gfCNCPoint5[14448] = {X 306.6871, Y 54.0357, Z -7.1667, A 0.000, B 0.000, C 0.000 }
gfCNCPoint5[14449] = {X 307.6171, Y 53.7103, Z -7.1667, A 0.000, B 0.000, C 0.000 }
gfCNCPoint5[14450] = {X 308.5962, Y 53.6000, Z -7.1667, A 0.000, B 0.000, C 0.000 }
gfCNCPoint5[14451] = {X 324.3107, Y 53.6000, Z -7.1667, A 0.000, B 0.000, C 0.000 }
gfCNCPoint5[14452] = {X 325.2898, Y 53.7103, Z -7.1667, A 0.000, B 0.000, C 0.000 }
gfCNCPoint5[14453] = {X 326.2198, Y 54.0357, Z -7.1667, A 0.000, B 0.000, C 0.000 }
gfCNCPoint5[14454] = {X 327.0540, Y 54.5599, Z -7.1667, A 0.000, B 0.000, C 0.000 }
gfCNCPoint5[14455] = {X 327.7507, Y 55.2566, Z -7.1667, A 0.000, B 0.000, C 0.000 }
gfCNCPoint5[14456] = {X 328.2750, Y 56.0909, Z -7.1667, A 0.000, B 0.000, C 0.000 }
gfCNCPoint5[14457] = {X 328.6004, Y 57.0209, Z -7.1667, A 0.000, B 0.000, C 0.000 }
gfCNCPoint5[14458] = {X 328.7107, Y 58.0000, Z -7.1667, A 0.000, B 0.000, C 0.000 }
gfCNCPoint5[14459] = {X 328.7107, Y 58.9362, Z -7.1667, A 0.000, B 0.000, C 0.000 }
gfCNCPoint5[14460] = {X 328.6172, Y 59.8190, Z -7.1667, A 0.000, B 0.000, C 0.000 }
gfCNCPoint5[14461] = {X 328.3499, Y 60.6656, Z -7.1667, A 0.000, B 0.000, C 0.000 }
gfCNCPoint5[14462] = {X 327.9194, Y 61.4419, Z -7.1667, A 0.000, B 0.000, C 0.000 }
gfCNCPoint5[14463] = {X 327.3430, Y 62.1171, Z -7.1667, A 0.000, B 0.000, C 0.000 }
gfCNCPoint5[14464] = {X 326.6437, Y 62.6640, Z -7.1667, A 0.000, B 0.000, C 0.000 }
gfCNCPoint5[14465] = {X 325.8496, Y 63.0607, Z -7.1667, A 0.000, B 0.000, C 0.000 }
gfCNCPoint5[14466] = {X 324.9923, Y 63.2915, Z -7.1667, A 0.000, B 0.000, C 0.000 }
gfCNCPoint5[14467] = {X 324.9942, Y 83.2293, Z -7.1667, A 0.000, B 0.000, C 0.000 }
gfCNCPoint5[14468] = {X 325.0078, Y 84.6142, Z -7.1667, A 0.000, B 0.000, C 0.000 }
gfCNCPoint5[14469] = {X 325.0827, Y 85.8241, Z -7.1667, A 0.000, B 0.000, C 0.000 }
gfCNCPoint5[14470] = {X 325.2965, Y 87.0173, Z -7.1667, A 0.000, B 0.000, C 0.000 }
gfCNCPoint5[14471] = {X 325.7310, Y 87.4224, Z -7.1667, A 0.000, B 0.000, C 0.000 }
gfCNCPoint5[14472] = {X 326.2477, Y 87.7156, Z -7.1667, A 0.000, B 0.000, C 0.000 }
gfCNCPoint5[14473] = {X 328.0176, Y 88.4226, Z -7.1667, A 0.000, B 0.000, C 0.000 }
gfCNCPoint5[14474] = {X 329.8594, Y 88.9123, Z -7.1667, A 0.000, B 0.000, C 0.000 }
gfCNCPoint5[14475] = {X 332.9373, Y 89.4644, Z -7.1667, A 0.000, B 0.000, C 0.000 }
gfCNCPoint5[14476] = {X 336.0431, Y 89.8280, Z -7.1667, A 0.000, B 0.000, C 0.000 }
gfCNCPoint5[14477] = {X 340.4120, Y 90.1221, Z -7.1667, A 0.000, B 0.000, C 0.000 }
gfCNCPoint5[14478] = {X 344.7882, Y 90.2759, Z -7.1667, A 0.000, B 0.000, C 0.000 }
gfCNCPoint5[14479] = {X 349.1670, Y 90.2890, Z -7.1667, A 0.000, B 0.000, C 0.000 }
gfCNCPoint5[14480] = {X 353.3143, Y 90.2206, Z -7.1667, A 0.000, B 0.000, C 0.000 }
gfCNCPoint5[14481] = {X 357.4564, Y 90.0018, Z -7.1667, A 0.000, B 0.000, C 0.000 }
gfCNCPoint5[14482] = {X 361.5878, Y 89.6328, Z -7.1667, A 0.000, B 0.000, C 0.000 }
gfCNCPoint5[14483] = {X 363.6656, Y 89.3462, Z -7.1667, A 0.000, B 0.000, C 0.000 }
gfCNCPoint5[14484] = {X 365.7243, Y 88.9447, Z -7.1667, A 0.000, B 0.000, C 0.000 }
gfCNCPoint5[14485] = {X 367.7576, Y 88.4298, Z -7.1667, A 0.000, B 0.000, C 0.000 }
gfCNCPoint5[14486] = {X 368.6806, Y 88.1197, Z -7.1667, A 0.000, B 0.000, C 0.000 }
gfCNCPoint5[14487] = {X 369.5629, Y 87.7078, Z -7.1667, A 0.000, B 0.000, C 0.000 }
gfCNCPoint5[14488] = {X 370.3933, Y 87.1992, Z -7.1667, A 0.000, B 0.000, C 0.000 }
gfCNCPoint5[14489] = {X 370.5198, Y 87.0673, Z -7.1667, A 0.000, B 0.000, C 0.000 }
gfCNCPoint5[14490] = {X 370.5851, Y 86.8966, Z -7.1667, A 0.000, B 0.000, C 0.000 }
gfCNCPoint5[14491] = {X 370.7755, Y 85.3680, Z -7.1667, A 0.000, B 0.000, C 0.000 }
gfCNCPoint5[14492] = {X 370.8391, Y 83.8288, Z -7.1667, A 0.000, B 0.000, C 0.000 }
gfCNCPoint5[14493] = {X 370.8379, Y 63.2810, Z -7.1667, A 0.000, B 0.000, C 0.000 }
gfCNCPoint5[14494] = {X 369.9788, Y 63.0556, Z -7.1667, A 0.000, B 0.000, C 0.000 }
gfCNCPoint5[14495] = {X 369.1826, Y 62.6623, Z -7.1667, A 0.000, B 0.000, C 0.000 }
gfCNCPoint5[14496] = {X 368.4815, Y 62.1171, Z -7.1667, A 0.000, B 0.000, C 0.000 }
gfCNCPoint5[14497] = {X 367.9042, Y 61.4423, Z -7.1667, A 0.000, B 0.000, C 0.000 }
gfCNCPoint5[14498] = {X 367.4741, Y 60.6652, Z -7.1667, A 0.000, B 0.000, C 0.000 }
gfCNCPoint5[14499] = {X 367.2089, Y 59.8176, Z -7.1667, A 0.000, B 0.000, C 0.000 }
gfCNCPoint5[14500] = {X 367.1193, Y 58.9341, Z -7.1667, A 0.000, B 0.000, C 0.000 }
gfCNCPoint5[14501] = {X 367.1193, Y 58.0000, Z -7.1667, A 0.000, B 0.000, C 0.000 }
gfCNCPoint5[14502] = {X 367.2296, Y 57.0209, Z -7.1667, A 0.000, B 0.000, C 0.000 }
gfCNCPoint5[14503] = {X 367.5550, Y 56.0909, Z -7.1667, A 0.000, B 0.000, C 0.000 }
gfCNCPoint5[14504] = {X 368.0792, Y 55.2566, Z -7.1667, A 0.000, B 0.000, C 0.000 }
gfCNCPoint5[14505] = {X 368.7759, Y 54.5599, Z -7.1667, A 0.000, B 0.000, C 0.000 }
gfCNCPoint5[14506] = {X 369.6102, Y 54.0357, Z -7.1667, A 0.000, B 0.000, C 0.000 }
gfCNCPoint5[14507] = {X 370.5402, Y 53.7103, Z -7.1667, A 0.000, B 0.000, C 0.000 }
gfCNCPoint5[14508] = {X 371.5193, Y 53.6000, Z -7.1667, A 0.000, B 0.000, C 0.000 }
gfCNCPoint5[14509] = {X 388.0597, Y 53.6000, Z -7.1667, A 0.000, B 0.000, C 0.000 }
gfCNCPoint5[14510] = {X 389.0388, Y 53.7103, Z -7.1667, A 0.000, B 0.000, C 0.000 }
gfCNCPoint5[14511] = {X 389.9688, Y 54.0357, Z -7.1667, A 0.000, B 0.000, C 0.000 }
gfCNCPoint5[14512] = {X 390.8030, Y 54.5599, Z -7.1667, A 0.000, B 0.000, C 0.000 }
gfCNCPoint5[14513] = {X 391.4997, Y 55.2566, Z -7.1667, A 0.000, B 0.000, C 0.000 }
gfCNCPoint5[14514] = {X 392.0239, Y 56.0909, Z -7.1667, A 0.000, B 0.000, C 0.000 }
gfCNCPoint5[14515] = {X 392.3494, Y 57.0209, Z -7.1667, A 0.000, B 0.000, C 0.000 }
gfCNCPoint5[14516] = {X 392.4597, Y 58.0000, Z -7.1667, A 0.000, B 0.000, C 0.000 }
gfCNCPoint5[14517] = {X 392.4595, Y 58.9704, Z -7.1667, A 0.000, B 0.000, C 0.000 }
gfCNCPoint5[14518] = {X 392.3419, Y 59.9454, Z -7.1667, A 0.000, B 0.000, C 0.000 }
gfCNCPoint5[14519] = {X 392.0109, Y 60.8701, Z -7.1667, A 0.000, B 0.000, C 0.000 }
gfCNCPoint5[14520] = {X 391.5686, Y 61.5895, Z -7.1667, A 0.000, B 0.000, C 0.000 }
gfCNCPoint5[14521] = {X 390.9977, Y 62.2117, Z -7.1667, A 0.000, B 0.000, C 0.000 }
gfCNCPoint5[14522] = {X 390.3190, Y 62.7141, Z -7.1667, A 0.000, B 0.000, C 0.000 }
gfCNCPoint5[14523] = {X 389.5572, Y 63.0784, Z -7.1667, A 0.000, B 0.000, C 0.000 }
gfCNCPoint5[14524] = {X 388.7400, Y 63.2913, Z -7.1667, A 0.000, B 0.000, C 0.000 }
gfCNCPoint5[14525] = {X 388.7400, Y 83.9247, Z -7.1667, A 0.000, B 0.000, C 0.000 }
gfCNCPoint5[14526] = {X 388.7379, Y 84.6149, Z -7.1667, A 0.000, B 0.000, C 0.000 }
gfCNCPoint5[14527] = {X 388.6777, Y 86.2800, Z -7.1667, A 0.000, B 0.000, C 0.000 }
gfCNCPoint5[14528] = {X 388.4725, Y 87.9334, Z -7.1667, A 0.000, B 0.000, C 0.000 }
gfCNCPoint5[14529] = {X 388.1239, Y 89.5626, Z -7.1667, A 0.000, B 0.000, C 0.000 }
gfCNCPoint5[14530] = {X 387.5878, Y 91.1605, Z -7.1667, A 0.000, B 0.000, C 0.000 }
gfCNCPoint5[14531] = {X 386.8330, Y 92.6676, Z -7.1667, A 0.000, B 0.000, C 0.000 }
gfCNCPoint5[14532] = {X 385.8745, Y 94.0540, Z -7.1667, A 0.000, B 0.000, C 0.000 }
gfCNCPoint5[14533] = {X 384.7313, Y 95.2924, Z -7.1667, A 0.000, B 0.000, C 0.000 }
gfCNCPoint5[14534] = {X 383.5035, Y 96.3481, Z -7.1667, A 0.000, B 0.000, C 0.000 }
gfCNCPoint5[14535] = {X 382.1889, Y 97.2937, Z -7.1667, A 0.000, B 0.000, C 0.000 }
gfCNCPoint5[14536] = {X 382.4521, Y 97.6951, Z -7.1667, A 0.000, B 0.000, C 0.000 }
gfCNCPoint5[14537] = {X 391.5259, Y 97.6951, Z -7.1667, A 0.000, B 0.000, C 0.000 }
gfCNCPoint5[14538] = {X 391.5259, Y 97.0659, Z -7.1667, A 0.000, B 0.000, C 0.000 }
gfCNCPoint5[14539] = {X 391.6193, Y 96.1159, Z -7.1667, A 0.000, B 0.000, C 0.000 }
gfCNCPoint5[14540] = {X 391.8959, Y 95.2021, Z -7.1667, A 0.000, B 0.000, C 0.000 }
gfCNCPoint5[14541] = {X 392.3450, Y 94.3598, Z -7.1667, A 0.000, B 0.000, C 0.000 }
gfCNCPoint5[14542] = {X 392.9496, Y 93.6209, Z -7.1667, A 0.000, B 0.000, C 0.000 }
gfCNCPoint5[14543] = {X 393.6864, Y 93.0139, Z -7.1667, A 0.000, B 0.000, C 0.000 }
gfCNCPoint5[14544] = {X 394.5273, Y 92.5620, Z -7.1667, A 0.000, B 0.000, C 0.000 }
gfCNCPoint5[14545] = {X 395.4401, Y 92.2825, Z -7.1667, A 0.000, B 0.000, C 0.000 }
gfCNCPoint5[14546] = {X 396.3899, Y 92.1860, Z -7.1667, A 0.000, B 0.000, C 0.000 }
gfCNCPoint5[14547] = {X 397.3090, Y 92.1443, Z -7.1667, A 0.000, B 0.000, C 0.000 }
gfCNCPoint5[14548] = {X 398.2250, Y 92.0575, Z -7.1667, A 0.000, B 0.000, C 0.000 }
gfCNCPoint5[14549] = {X 398.7531, Y 91.9291, Z -7.1667, A 0.000, B 0.000, C 0.000 }
gfCNCPoint5[14550] = {X 399.2394, Y 91.6865, Z -7.1667, A 0.000, B 0.000, C 0.000 }
gfCNCPoint5[14551] = {X 426.8261, Y 74.0196, Z -7.1667, A 0.000, B 0.000, C 0.000 }
gfCNCPoint5[14552] = {X 403.5510, Y 64.8882, Z -7.1667, A 0.000, B 0.000, C 0.000 }
gfCNCPoint5[14553] = {X 402.0098, Y 64.3725, Z -7.1667, A 0.000, B 0.000, C 0.000 }
gfCNCPoint5[14554] = {X 400.4236, Y 64.0186, Z -7.1667, A 0.000, B 0.000, C 0.000 }
gfCNCPoint5[14555] = {X 398.8190, Y 73.4835, Z -7.1667, A 0.000, B 0.000, C 0.000 }
gfCNCPoint5[14556] = {X 398.8183, Y 80.5563, Z -7.1667, A 0.000, B 0.000, C 0.000 }
gfCNCPoint5[14557] = {X 405.8022, Y 76.0837, Z -7.1667, A 0.000, B 0.000, C 0.000 }
gfCNCPoint5[14558] = {X 400.0393, Y 73.8228, Z -7.1667, A 0.000, B 0.000, C 0.000 }
gfCNCPoint5[14559] = {X 399.4379, Y 73.6216, Z -7.1667, A 0.000, B 0.000, C 0.000 }
gfCNCPoint5[14560] = {X 398.8190, Y 73.4835, Z -7.1667, A 0.000, B 0.000, C 0.000 }
gfCNCPoint5[14561] = {X 399.2202, Y 71.1173, Z -7.1667, A 0.000, B 0.000, C 0.000 }
gfCNCPoint5[14562] = {X 398.7493, Y 71.0509, Z -7.1667, A 0.000, B 0.000, C 0.000 }
gfCNCPoint5[14563] = {X 398.2755, Y 71.0108, Z -7.1667, A 0.000, B 0.000, C 0.000 }
gfCNCPoint5[14564] = {X 397.3438, Y 70.9529, Z -7.1667, A 0.000, B 0.000, C 0.000 }
gfCNCPoint5[14565] = {X 396.4193, Y 70.8233, Z -7.1667, A 0.000, B 0.000, C 0.000 }
gfCNCPoint5[14566] = {X 396.4180, Y 84.5897, Z -7.1667, A 0.000, B 0.000, C 0.000 }
gfCNCPoint5[14567] = {X 396.4178, Y 84.9436, Z -7.1667, A 0.000, B 0.000, C 0.000 }
gfCNCPoint5[14568] = {X 411.0581, Y 75.5677, Z -7.1667, A 0.000, B 0.000, C 0.000 }
gfCNCPoint5[14569] = {X 400.9172, Y 71.5892, Z -7.1667, A 0.000, B 0.000, C 0.000 }
gfCNCPoint5[14570] = {X 400.0809, Y 71.3094, Z -7.1667, A 0.000, B 0.000, C 0.000 }
gfCNCPoint5[14571] = {X 399.2202, Y 71.1173, Z -7.1667, A 0.000, B 0.000, C 0.000 }
gfCNCPoint5[14572] = {X 399.6213, Y 68.7510, Z -7.1667, A 0.000, B 0.000, C 0.000 }
gfCNCPoint5[14573] = {X 398.9961, Y 68.6635, Z -7.1667, A 0.000, B 0.000, C 0.000 }
gfCNCPoint5[14574] = {X 398.3668, Y 68.6122, Z -7.1667, A 0.000, B 0.000, C 0.000 }
gfCNCPoint5[14575] = {X 397.6025, Y 68.5668, Z -7.1667, A 0.000, B 0.000, C 0.000 }
gfCNCPoint5[14576] = {X 396.8441, Y 68.4612, Z -7.1667, A 0.000, B 0.000, C 0.000 }
gfCNCPoint5[14577] = {X 395.3939, Y 68.0824, Z -7.1667, A 0.000, B 0.000, C 0.000 }
gfCNCPoint5[14578] = {X 394.0196, Y 67.4844, Z -7.1667, A 0.000, B 0.000, C 0.000 }
gfCNCPoint5[14579] = {X 394.0180, Y 84.5973, Z -7.1667, A 0.000, B 0.000, C 0.000 }
gfCNCPoint5[14580] = {X 394.0185, Y 84.7621, Z -7.1667, A 0.000, B 0.000, C 0.000 }
gfCNCPoint5[14581] = {X 394.0179, Y 84.9270, Z -7.1667, A 0.000, B 0.000, C 0.000 }
gfCNCPoint5[14582] = {X 393.9676, Y 86.3327, Z -7.1667, A 0.000, B 0.000, C 0.000 }
gfCNCPoint5[14583] = {X 393.8362, Y 87.7333, Z -7.1667, A 0.000, B 0.000, C 0.000 }
gfCNCPoint5[14584] = {X 395.0679, Y 87.4789, Z -7.1667, A 0.000, B 0.000, C 0.000 }
gfCNCPoint5[14585] = {X 396.3222, Y 87.3863, Z -7.1667, A 0.000, B 0.000, C 0.000 }
gfCNCPoint5[14586] = {X 396.7204, Y 87.3714, Z -7.1667, A 0.000, B 0.000, C 0.000 }
gfCNCPoint5[14587] = {X 397.1179, Y 87.3452, Z -7.1667, A 0.000, B 0.000, C 0.000 }
gfCNCPoint5[14588] = {X 416.3141, Y 75.0517, Z -7.1667, A 0.000, B 0.000, C 0.000 }
gfCNCPoint5[14589] = {X 401.7952, Y 69.3555, Z -7.1667, A 0.000, B 0.000, C 0.000 }
gfCNCPoint5[14590] = {X 400.7239, Y 68.9971, Z -7.1667, A 0.000, B 0.000, C 0.000 }
gfCNCPoint5[14591] = {X 399.6213, Y 68.7510, Z -7.1667, A 0.000, B 0.000, C 0.000 }
gfCNCPoint5[14592] = {X 400.0225, Y 66.3848, Z -7.1667, A 0.000, B 0.000, C 0.000 }
gfCNCPoint5[14593] = {X 399.2382, Y 66.2757, Z -7.1667, A 0.000, B 0.000, C 0.000 }
gfCNCPoint5[14594] = {X 398.4488, Y 66.2132, Z -7.1667, A 0.000, B 0.000, C 0.000 }
gfCNCPoint5[14595] = {X 397.3046, Y 66.1054, Z -7.1667, A 0.000, B 0.000, C 0.000 }
gfCNCPoint5[14596] = {X 396.1916, Y 65.8188, Z -7.1667, A 0.000, B 0.000, C 0.000 }
gfCNCPoint5[14597] = {X 395.1376, Y 65.3607, Z -7.1667, A 0.000, B 0.000, C 0.000 }
gfCNCPoint5[14598] = {X 394.1689, Y 64.7424, Z -7.1667, A 0.000, B 0.000, C 0.000 }
gfCNCPoint5[14599] = {X 393.3095, Y 63.9793, Z -7.1667, A 0.000, B 0.000, C 0.000 }
gfCNCPoint5[14600] = {X 392.5128, Y 64.6963, Z -7.1667, A 0.000, B 0.000, C 0.000 }
gfCNCPoint5[14601] = {X 391.6198, Y 65.2889, Z -7.1667, A 0.000, B 0.000, C 0.000 }
gfCNCPoint5[14602] = {X 391.6180, Y 84.6054, Z -7.1667, A 0.000, B 0.000, C 0.000 }
gfCNCPoint5[14603] = {X 391.5819, Y 86.0254, Z -7.1667, A 0.000, B 0.000, C 0.000 }
gfCNCPoint5[14604] = {X 391.4541, Y 87.4402, Z -7.1667, A 0.000, B 0.000, C 0.000 }
gfCNCPoint5[14605] = {X 391.2298, Y 88.8724, Z -7.1667, A 0.000, B 0.000, C 0.000 }
gfCNCPoint5[14606] = {X 390.9114, Y 90.2866, Z -7.1667, A 0.000, B 0.000, C 0.000 }
gfCNCPoint5[14607] = {X 390.3349, Y 92.0503, Z -7.1667, A 0.000, B 0.000, C 0.000 }
gfCNCPoint5[14608] = {X 389.5433, Y 93.7285, Z -7.1667, A 0.000, B 0.000, C 0.000 }
gfCNCPoint5[14609] = {X 388.5489, Y 95.2951, Z -7.1667, A 0.000, B 0.000, C 0.000 }
gfCNCPoint5[14610] = {X 389.3446, Y 95.2951, Z -7.1667, A 0.000, B 0.000, C 0.000 }
gfCNCPoint5[14611] = {X 389.7639, Y 94.0857, Z -7.1667, A 0.000, B 0.000, C 0.000 }
gfCNCPoint5[14612] = {X 390.3886, Y 92.9683, Z -7.1667, A 0.000, B 0.000, C 0.000 }
gfCNCPoint5[14613] = {X 391.1994, Y 91.9777, Z -7.1667, A 0.000, B 0.000, C 0.000 }
gfCNCPoint5[14614] = {X 392.1711, Y 91.1444, Z -7.1667, A 0.000, B 0.000, C 0.000 }
gfCNCPoint5[14615] = {X 393.2738, Y 90.4942, Z -7.1667, A 0.000, B 0.000, C 0.000 }
gfCNCPoint5[14616] = {X 394.4733, Y 90.0472, Z -7.1667, A 0.000, B 0.000, C 0.000 }
gfCNCPoint5[14617] = {X 395.4072, Y 89.8548, Z -7.1667, A 0.000, B 0.000, C 0.000 }
gfCNCPoint5[14618] = {X 396.3583, Y 89.7861, Z -7.1667, A 0.000, B 0.000, C 0.000 }
gfCNCPoint5[14619] = {X 397.1424, Y 89.7501, Z -7.1667, A 0.000, B 0.000, C 0.000 }
gfCNCPoint5[14620] = {X 397.9239, Y 89.6764, Z -7.1667, A 0.000, B 0.000, C 0.000 }
gfCNCPoint5[14621] = {X 417.6084, Y 77.0728, Z -7.1667, A 0.000, B 0.000, C 0.000 }
gfCNCPoint5[14622] = {X 421.5701, Y 74.5357, Z -7.1667, A 0.000, B 0.000, C 0.000 }
gfCNCPoint5[14623] = {X 402.6731, Y 67.1218, Z -7.1667, A 0.000, B 0.000, C 0.000 }
gfCNCPoint5[14624] = {X 401.3668, Y 66.6848, Z -7.1667, A 0.000, B 0.000, C 0.000 }
gfCNCPoint5[14625] = {X 400.0225, Y 66.3848, Z -7.1667, A 0.000, B 0.000, C 0.000 }
gfCNCPoint5[14626] = {X 400.4236, Y 64.0186, Z -7.1667, A 0.000, B 0.000, C 0.000 }
gfCNCPoint5[14627] = {X 399.4750, Y 63.8873, Z -7.1667, A 0.000, B 0.000, C 0.000 }
gfCNCPoint5[14628] = {X 398.5200, Y 63.8139, Z -7.1667, A 0.000, B 0.000, C 0.000 }
gfCNCPoint5[14629] = {X 397.5544, Y 63.7098, Z -7.1667, A 0.000, B 0.000, C 0.000 }
gfCNCPoint5[14630] = {X 396.6285, Y 63.4165, Z -7.1667, A 0.000, B 0.000, C 0.000 }
gfCNCPoint5[14631] = {X 395.7791, Y 62.9457, Z -7.1667, A 0.000, B 0.000, C 0.000 }
gfCNCPoint5[14632] = {X 395.0397, Y 62.3160, Z -7.1667, A 0.000, B 0.000, C 0.000 }
gfCNCPoint5[14633] = {X 394.4660, Y 61.5934, Z -7.1667, A 0.000, B 0.000, C 0.000 }
gfCNCPoint5[14634] = {X 394.0386, Y 60.7757, Z -7.1667, A 0.000, B 0.000, C 0.000 }
gfCNCPoint5[14635] = {X 393.7727, Y 59.8922, Z -7.1667, A 0.000, B 0.000, C 0.000 }
gfCNCPoint5[14636] = {X 393.6779, Y 58.9744, Z -7.1667, A 0.000, B 0.000, C 0.000 }
gfCNCPoint5[14637] = {X 393.6777, Y 58.0000, Z -7.1667, A 0.000, B 0.000, C 0.000 }
gfCNCPoint5[14638] = {X 393.7668, Y 57.0718, Z -7.1667, A 0.000, B 0.000, C 0.000 }
gfCNCPoint5[14639] = {X 394.0309, Y 56.1774, Z -7.1667, A 0.000, B 0.000, C 0.000 }
gfCNCPoint5[14640] = {X 394.4602, Y 55.3496, Z -7.1667, A 0.000, B 0.000, C 0.000 }
gfCNCPoint5[14641] = {X 395.0391, Y 54.6186, Z -7.1667, A 0.000, B 0.000, C 0.000 }
gfCNCPoint5[14642] = {X 395.7864, Y 53.9833, Z -7.1667, A 0.000, B 0.000, C 0.000 }
gfCNCPoint5[14643] = {X 396.6455, Y 53.5102, Z -7.1667, A 0.000, B 0.000, C 0.000 }
gfCNCPoint5[14644] = {X 397.5819, Y 53.2186, Z -7.1667, A 0.000, B 0.000, C 0.000 }
gfCNCPoint5[14645] = {X 398.5577, Y 53.1200, Z -7.1667, A 0.000, B 0.000, C 0.000 }
gfCNCPoint5[14646] = {X 419.4886, Y 53.1200, Z -7.1667, A 0.000, B 0.000, C 0.000 }
gfCNCPoint5[14647] = {X 420.5533, Y 53.2376, Z -7.1667, A 0.000, B 0.000, C 0.000 }
gfCNCPoint5[14648] = {X 421.5667, Y 53.5846, Z -7.1667, A 0.000, B 0.000, C 0.000 }
gfCNCPoint5[14649] = {X 422.4800, Y 54.1443, Z -7.1667, A 0.000, B 0.000, C 0.000 }
gfCNCPoint5[14650] = {X 423.2491, Y 54.8899, Z -7.1667, A 0.000, B 0.000, C 0.000 }
gfCNCPoint5[14651] = {X 423.8371, Y 55.7852, Z -7.1667, A 0.000, B 0.000, C 0.000 }
gfCNCPoint5[14652] = {X 424.2155, Y 56.7873, Z -7.1667, A 0.000, B 0.000, C 0.000 }
gfCNCPoint5[14653] = {X 424.3662, Y 57.8478, Z -7.1667, A 0.000, B 0.000, C 0.000 }
gfCNCPoint5[14654] = {X 429.8191, Y 59.9722, Z -7.1667, A 0.000, B 0.000, C 0.000 }
gfCNCPoint5[14655] = {X 457.2980, Y 70.8751, Z -7.1667, A 0.000, B 0.000, C 0.000 }
gfCNCPoint5[14656] = {X 457.2983, Y 63.6739, Z -7.1667, A 0.000, B 0.000, C 0.000 }
gfCNCPoint5[14657] = {X 456.2903, Y 63.3054, Z -7.1667, A 0.000, B 0.000, C 0.000 }
gfCNCPoint5[14658] = {X 455.3872, Y 62.7254, Z -7.1667, A 0.000, B 0.000, C 0.000 }
gfCNCPoint5[14659] = {X 454.6327, Y 61.9621, Z -7.1667, A 0.000, B 0.000, C 0.000 }
gfCNCPoint5[14660] = {X 454.0633, Y 61.0524, Z -7.1667, A 0.000, B 0.000, C 0.000 }
gfCNCPoint5[14661] = {X 453.7066, Y 60.0401, Z -7.1667, A 0.000, B 0.000, C 0.000 }
gfCNCPoint5[14662] = {X 453.5798, Y 58.9744, Z -7.1667, A 0.000, B 0.000, C 0.000 }
gfCNCPoint5[14663] = {X 453.5796, Y 58.0000, Z -7.1667, A 0.000, B 0.000, C 0.000 }
gfCNCPoint5[14664] = {X 453.6734, Y 57.0480, Z -7.1667, A 0.000, B 0.000, C 0.000 }
gfCNCPoint5[14665] = {X 453.9511, Y 56.1325, Z -7.1667, A 0.000, B 0.000, C 0.000 }
gfCNCPoint5[14666] = {X 454.4020, Y 55.2888, Z -7.1667, A 0.000, B 0.000, C 0.000 }
gfCNCPoint5[14667] = {X 455.0089, Y 54.5493, Z -7.1667, A 0.000, B 0.000, C 0.000 }
gfCNCPoint5[14668] = {X 455.7484, Y 53.9424, Z -7.1667, A 0.000, B 0.000, C 0.000 }
gfCNCPoint5[14669] = {X 456.5921, Y 53.4915, Z -7.1667, A 0.000, B 0.000, C 0.000 }
gfCNCPoint5[14670] = {X 457.5076, Y 53.2138, Z -7.1667, A 0.000, B 0.000, C 0.000 }
gfCNCPoint5[14671] = {X 458.4596, Y 53.1200, Z -7.1667, A 0.000, B 0.000, C 0.000 }
gfCNCPoint5[14672] = {X 475.0000, Y 53.1200, Z -7.1667, A 0.000, B 0.000, C 0.000 }
gfCNCPoint5[14673] = {X 475.9520, Y 53.2138, Z -7.1667, A 0.000, B 0.000, C 0.000 }
gfCNCPoint5[14674] = {X 476.8675, Y 53.4915, Z -7.1667, A 0.000, B 0.000, C 0.000 }
gfCNCPoint5[14675] = {X 477.7112, Y 53.9424, Z -7.1667, A 0.000, B 0.000, C 0.000 }
gfCNCPoint5[14676] = {X 478.4507, Y 54.5493, Z -7.1667, A 0.000, B 0.000, C 0.000 }
gfCNCPoint5[14677] = {X 479.0576, Y 55.2888, Z -7.1667, A 0.000, B 0.000, C 0.000 }
gfCNCPoint5[14678] = {X 479.5085, Y 56.1325, Z -7.1667, A 0.000, B 0.000, C 0.000 }
gfCNCPoint5[14679] = {X 479.7862, Y 57.0480, Z -7.1667, A 0.000, B 0.000, C 0.000 }
gfCNCPoint5[14680] = {X 479.8800, Y 58.0000, Z -7.1667, A 0.000, B 0.000, C 0.000 }
gfCNCPoint5[14681] = {X 479.8798, Y 58.9744, Z -7.1667, A 0.000, B 0.000, C 0.000 }
gfCNCPoint5[14682] = {X 479.7530, Y 60.0402, Z -7.1667, A 0.000, B 0.000, C 0.000 }
gfCNCPoint5[14683] = {X 479.3962, Y 61.0525, Z -7.1667, A 0.000, B 0.000, C 0.000 }
gfCNCPoint5[14684] = {X 478.8268, Y 61.9623, Z -7.1667, A 0.000, B 0.000, C 0.000 }
gfCNCPoint5[14685] = {X 478.0722, Y 62.7256, Z -7.1667, A 0.000, B 0.000, C 0.000 }
gfCNCPoint5[14686] = {X 477.1691, Y 63.3055, Z -7.1667, A 0.000, B 0.000, C 0.000 }
gfCNCPoint5[14687] = {X 476.1610, Y 63.6739, Z -7.1667, A 0.000, B 0.000, C 0.000 }
gfCNCPoint5[14688] = {X 476.1614, Y 92.3307, Z -7.1667, A 0.000, B 0.000, C 0.000 }
gfCNCPoint5[14689] = {X 476.3600, Y 92.3888, Z -7.1667, A 0.000, B 0.000, C 0.000 }
gfCNCPoint5[14690] = {X 476.5570, Y 92.4517, Z -7.1667, A 0.000, B 0.000, C 0.000 }
gfCNCPoint5[14691] = {X 477.4766, Y 92.8687, Z -7.1667, A 0.000, B 0.000, C 0.000 }
gfCNCPoint5[14692] = {X 478.2902, Y 93.4667, Z -7.1667, A 0.000, B 0.000, C 0.000 }
gfCNCPoint5[14693] = {X 478.9626, Y 94.2200, Z -7.1667, A 0.000, B 0.000, C 0.000 }
gfCNCPoint5[14694] = {X 479.4648, Y 95.0960, Z -7.1667, A 0.000, B 0.000, C 0.000 }
gfCNCPoint5[14695] = {X 479.7751, Y 96.0569, Z -7.1667, A 0.000, B 0.000, C 0.000 }
gfCNCPoint5[14696] = {X 479.8800, Y 97.0611, Z -7.1667, A 0.000, B 0.000, C 0.000 }
gfCNCPoint5[14697] = {X 479.8800, Y 97.6951, Z -7.1667, A 0.000, B 0.000, C 0.000 }
gfCNCPoint5[14698] = {X 479.4000, Y 97.6951, Z -7.1667, A 0.000, B 0.000, C 0.000 }
gfCNCPoint5[14699] = {X 479.4000, Y 98.0000, Z -7.1667, A 0.000, B 0.000, C 0.000 }
gfCNCPoint5[14700] = {X 479.2897, Y 98.9791, Z -7.1667, A 0.000, B 0.000, C 0.000 }
gfCNCPoint5[14701] = {X 478.9643, Y 99.9091, Z -7.1667, A 0.000, B 0.000, C 0.000 }
gfCNCPoint5[14702] = {X 478.4401, Y 100.7434, Z -7.1667, A 0.000, B 0.000, C 0.000 }
gfCNCPoint5[14703] = {X 477.7434, Y 101.4401, Z -7.1667, A 0.000, B 0.000, C 0.000 }
gfCNCPoint5[14704] = {X 476.9091, Y 101.9643, Z -7.1667, A 0.000, B 0.000, C 0.000 }
gfCNCPoint5[14705] = {X 475.9791, Y 102.2897, Z -7.1667, A 0.000, B 0.000, C 0.000 }
gfCNCPoint5[14706] = {X 475.0000, Y 102.4000, Z -7.1667, A 0.000, B 0.000, C 0.000 }
gfCNCPoint5[14707] = {X 458.4596, Y 102.4000, Z -7.1667, A 0.000, B 0.000, C 0.000 }
gfCNCPoint5[14708] = {X 457.4805, Y 102.2897, Z -7.1667, A 0.000, B 0.000, C 0.000 }
gfCNCPoint5[14709] = {X 456.5505, Y 101.9643, Z -7.1667, A 0.000, B 0.000, C 0.000 }
gfCNCPoint5[14710] = {X 455.7162, Y 101.4401, Z -7.1667, A 0.000, B 0.000, C 0.000 }
gfCNCPoint5[14711] = {X 455.0195, Y 100.7434, Z -7.1667, A 0.000, B 0.000, C 0.000 }
gfCNCPoint5[14712] = {X 454.4953, Y 99.9091, Z -7.1667, A 0.000, B 0.000, C 0.000 }
gfCNCPoint5[14713] = {X 454.1699, Y 98.9791, Z -7.1667, A 0.000, B 0.000, C 0.000 }
gfCNCPoint5[14714] = {X 454.0596, Y 98.0000, Z -7.1667, A 0.000, B 0.000, C 0.000 }
gfCNCPoint5[14715] = {X 454.0596, Y 97.0659, Z -7.1667, A 0.000, B 0.000, C 0.000 }
gfCNCPoint5[14716] = {X 454.1492, Y 96.1826, Z -7.1667, A 0.000, B 0.000, C 0.000 }
gfCNCPoint5[14717] = {X 454.4143, Y 95.3353, Z -7.1667, A 0.000, B 0.000, C 0.000 }
gfCNCPoint5[14718] = {X 454.8440, Y 94.5584, Z -7.1667, A 0.000, B 0.000, C 0.000 }
gfCNCPoint5[14719] = {X 455.4210, Y 93.8836, Z -7.1667, A 0.000, B 0.000, C 0.000 }
gfCNCPoint5[14720] = {X 456.1217, Y 93.3384, Z -7.1667, A 0.000, B 0.000, C 0.000 }
gfCNCPoint5[14721] = {X 456.9176, Y 92.9450, Z -7.1667, A 0.000, B 0.000, C 0.000 }
gfCNCPoint5[14722] = {X 457.7763, Y 92.7193, Z -7.1667, A 0.000, B 0.000, C 0.000 }
gfCNCPoint5[14723] = {X 457.7763, Y 85.6495, Z -7.1667, A 0.000, B 0.000, C 0.000 }
gfCNCPoint5[14724] = {X 444.8692, Y 80.5899, Z -7.1667, A 0.000, B 0.000, C 0.000 }
gfCNCPoint5[14725] = {X 420.1044, Y 96.6318, Z -7.1667, A 0.000, B 0.000, C 0.000 }
gfCNCPoint5[14726] = {X 420.1067, Y 97.0659, Z -7.1667, A 0.000, B 0.000, C 0.000 }
gfCNCPoint5[14727] = {X 420.1067, Y 98.0000, Z -7.1667, A 0.000, B 0.000, C 0.000 }
gfCNCPoint5[14728] = {X 419.9964, Y 98.9791, Z -7.1667, A 0.000, B 0.000, C 0.000 }
gfCNCPoint5[14729] = {X 419.6710, Y 99.9091, Z -7.1667, A 0.000, B 0.000, C 0.000 }
gfCNCPoint5[14730] = {X 419.1468, Y 100.7434, Z -7.1667, A 0.000, B 0.000, C 0.000 }
gfCNCPoint5[14731] = {X 418.4501, Y 101.4401, Z -7.1667, A 0.000, B 0.000, C 0.000 }
gfCNCPoint5[14732] = {X 417.6158, Y 101.9643, Z -7.1667, A 0.000, B 0.000, C 0.000 }
gfCNCPoint5[14733] = {X 416.6858, Y 102.2897, Z -7.1667, A 0.000, B 0.000, C 0.000 }
gfCNCPoint5[14734] = {X 415.7067, Y 102.4000, Z -7.1667, A 0.000, B 0.000, C 0.000 }
gfCNCPoint5[14735] = {X 396.4059, Y 102.4000, Z -7.1667, A 0.000, B 0.000, C 0.000 }
gfCNCPoint5[14736] = {X 395.4269, Y 102.2897, Z -7.1667, A 0.000, B 0.000, C 0.000 }
gfCNCPoint5[14737] = {X 394.4969, Y 101.9643, Z -7.1667, A 0.000, B 0.000, C 0.000 }
gfCNCPoint5[14738] = {X 393.6626, Y 101.4401, Z -7.1667, A 0.000, B 0.000, C 0.000 }
gfCNCPoint5[14739] = {X 392.9659, Y 100.7434, Z -7.1667, A 0.000, B 0.000, C 0.000 }
gfCNCPoint5[14740] = {X 392.4417, Y 99.9091, Z -7.1667, A 0.000, B 0.000, C 0.000 }
gfCNCPoint5[14741] = {X 392.1163, Y 98.9791, Z -7.1667, A 0.000, B 0.000, C 0.000 }
gfCNCPoint5[14742] = {X 392.0059, Y 98.0000, Z -7.1667, A 0.000, B 0.000, C 0.000 }
gfCNCPoint5[14743] = {X 392.0059, Y 97.0659, Z -7.1667, A 0.000, B 0.000, C 0.000 }
gfCNCPoint5[14744] = {X 392.1159, Y 96.0883, Z -7.1667, A 0.000, B 0.000, C 0.000 }
gfCNCPoint5[14745] = {X 392.4404, Y 95.1595, Z -7.1667, A 0.000, B 0.000, C 0.000 }
gfCNCPoint5[14746] = {X 392.9631, Y 94.3261, Z -7.1667, A 0.000, B 0.000, C 0.000 }
gfCNCPoint5[14747] = {X 393.6579, Y 93.6296, Z -7.1667, A 0.000, B 0.000, C 0.000 }
gfCNCPoint5[14748] = {X 394.4902, Y 93.1049, Z -7.1667, A 0.000, B 0.000, C 0.000 }
gfCNCPoint5[14749] = {X 395.4182, Y 92.7782, Z -7.1667, A 0.000, B 0.000, C 0.000 }
gfCNCPoint5[14750] = {X 396.3955, Y 92.6659, Z -7.1667, A 0.000, B 0.000, C 0.000 }
gfCNCPoint5[14751] = {X 397.3413, Y 92.6232, Z -7.1667, A 0.000, B 0.000, C 0.000 }
gfCNCPoint5[14752] = {X 398.2838, Y 92.5339, Z -7.1667, A 0.000, B 0.000, C 0.000 }
gfCNCPoint5[14753] = {X 398.9171, Y 92.3802, Z -7.1667, A 0.000, B 0.000, C 0.000 }
gfCNCPoint5[14754] = {X 399.5003, Y 92.0894, Z -7.1667, A 0.000, B 0.000, C 0.000 }
gfCNCPoint5[14755] = {X 404.0998, Y 89.1252, Z -7.1667, A 0.000, B 0.000, C 0.000 }
gfCNCPoint5[14756] = {X 427.8779, Y 73.9167, Z -7.1667, A 0.000, B 0.000, C 0.000 }
gfCNCPoint5[14757] = {X 403.7263, Y 64.4413, Z -7.1667, A 0.000, B 0.000, C 0.000 }
gfCNCPoint5[14758] = {X 402.0391, Y 63.8828, Z -7.1667, A 0.000, B 0.000, C 0.000 }
gfCNCPoint5[14759] = {X 400.3009, Y 63.5122, Z -7.1667, A 0.000, B 0.000, C 0.000 }
gfCNCPoint5[14760] = {X 398.5327, Y 63.3340, Z -7.1667, A 0.000, B 0.000, C 0.000 }
gfCNCPoint5[14761] = {X 397.5577, Y 63.2189, Z -7.1667, A 0.000, B 0.000, C 0.000 }
gfCNCPoint5[14762] = {X 396.6325, Y 62.8905, Z -7.1667, A 0.000, B 0.000, C 0.000 }
gfCNCPoint5[14763] = {X 395.8032, Y 62.3652, Z -7.1667, A 0.000, B 0.000, C 0.000 }
gfCNCPoint5[14764] = {X 395.1110, Y 61.6690, Z -7.1667, A 0.000, B 0.000, C 0.000 }
gfCNCPoint5[14765] = {X 394.5904, Y 60.8367, Z -7.1667, A 0.000, B 0.000, C 0.000 }
gfCNCPoint5[14766] = {X 394.2672, Y 59.9097, Z -7.1667, A 0.000, B 0.000, C 0.000 }
gfCNCPoint5[14767] = {X 394.1577, Y 58.9341, Z -7.1667, A 0.000, B 0.000, C 0.000 }
gfCNCPoint5[14768] = {X 394.1577, Y 58.0000, Z -7.1667, A 0.000, B 0.000, C 0.000 }
gfCNCPoint5[14769] = {X 394.2680, Y 57.0209, Z -7.1667, A 0.000, B 0.000, C 0.000 }
gfCNCPoint5[14770] = {X 394.5935, Y 56.0909, Z -7.1667, A 0.000, B 0.000, C 0.000 }
gfCNCPoint5[14771] = {X 395.1177, Y 55.2566, Z -7.1667, A 0.000, B 0.000, C 0.000 }
gfCNCPoint5[14772] = {X 395.8144, Y 54.5599, Z -7.1667, A 0.000, B 0.000, C 0.000 }
gfCNCPoint5[14773] = {X 396.6486, Y 54.0357, Z -7.1667, A 0.000, B 0.000, C 0.000 }
gfCNCPoint5[14774] = {X 397.5786, Y 53.7103, Z -7.1667, A 0.000, B 0.000, C 0.000 }
gfCNCPoint5[14775] = {X 398.5577, Y 53.6000, Z -7.1667, A 0.000, B 0.000, C 0.000 }
gfCNCPoint5[14776] = {X 419.4886, Y 53.6000, Z -7.1667, A 0.000, B 0.000, C 0.000 }
gfCNCPoint5[14777] = {X 420.4677, Y 53.7103, Z -7.1667, A 0.000, B 0.000, C 0.000 }
gfCNCPoint5[14778] = {X 421.3977, Y 54.0357, Z -7.1667, A 0.000, B 0.000, C 0.000 }
gfCNCPoint5[14779] = {X 422.2320, Y 54.5599, Z -7.1667, A 0.000, B 0.000, C 0.000 }
gfCNCPoint5[14780] = {X 422.9287, Y 55.2566, Z -7.1667, A 0.000, B 0.000, C 0.000 }
gfCNCPoint5[14781] = {X 423.4529, Y 56.0909, Z -7.1667, A 0.000, B 0.000, C 0.000 }
gfCNCPoint5[14782] = {X 423.7783, Y 57.0209, Z -7.1667, A 0.000, B 0.000, C 0.000 }
gfCNCPoint5[14783] = {X 423.8886, Y 58.0000, Z -7.1667, A 0.000, B 0.000, C 0.000 }
gfCNCPoint5[14784] = {X 423.8886, Y 58.1769, Z -7.1667, A 0.000, B 0.000, C 0.000 }
gfCNCPoint5[14785] = {X 429.6420, Y 60.4184, Z -7.1667, A 0.000, B 0.000, C 0.000 }
gfCNCPoint5[14786] = {X 457.7780, Y 71.5820, Z -7.1667, A 0.000, B 0.000, C 0.000 }
gfCNCPoint5[14787] = {X 457.7783, Y 63.2810, Z -7.1667, A 0.000, B 0.000, C 0.000 }
gfCNCPoint5[14788] = {X 456.9193, Y 63.0556, Z -7.1667, A 0.000, B 0.000, C 0.000 }
gfCNCPoint5[14789] = {X 456.1230, Y 62.6623, Z -7.1667, A 0.000, B 0.000, C 0.000 }
gfCNCPoint5[14790] = {X 455.4219, Y 62.1172, Z -7.1667, A 0.000, B 0.000, C 0.000 }
gfCNCPoint5[14791] = {X 454.8445, Y 61.4423, Z -7.1667, A 0.000, B 0.000, C 0.000 }
gfCNCPoint5[14792] = {X 454.4145, Y 60.6652, Z -7.1667, A 0.000, B 0.000, C 0.000 }
gfCNCPoint5[14793] = {X 454.1492, Y 59.8176, Z -7.1667, A 0.000, B 0.000, C 0.000 }
gfCNCPoint5[14794] = {X 454.0596, Y 58.9341, Z -7.1667, A 0.000, B 0.000, C 0.000 }
gfCNCPoint5[14795] = {X 454.0596, Y 58.0000, Z -7.1667, A 0.000, B 0.000, C 0.000 }
gfCNCPoint5[14796] = {X 454.1699, Y 57.0209, Z -7.1667, A 0.000, B 0.000, C 0.000 }
gfCNCPoint5[14797] = {X 454.4953, Y 56.0909, Z -7.1667, A 0.000, B 0.000, C 0.000 }
gfCNCPoint5[14798] = {X 455.0195, Y 55.2566, Z -7.1667, A 0.000, B 0.000, C 0.000 }
gfCNCPoint5[14799] = {X 455.7162, Y 54.5599, Z -7.1667, A 0.000, B 0.000, C 0.000 }
gfCNCPoint5[14800] = {X 456.5505, Y 54.0357, Z -7.1667, A 0.000, B 0.000, C 0.000 }
gfCNCPoint5[14801] = {X 457.4805, Y 53.7103, Z -7.1667, A 0.000, B 0.000, C 0.000 }
gfCNCPoint5[14802] = {X 458.4596, Y 53.6000, Z -7.1667, A 0.000, B 0.000, C 0.000 }
gfCNCPoint5[14803] = {X 475.0000, Y 53.6000, Z -7.1667, A 0.000, B 0.000, C 0.000 }
gfCNCPoint5[14804] = {X 475.9791, Y 53.7103, Z -7.1667, A 0.000, B 0.000, C 0.000 }
gfCNCPoint5[14805] = {X 476.9091, Y 54.0357, Z -7.1667, A 0.000, B 0.000, C 0.000 }
gfCNCPoint5[14806] = {X 477.7434, Y 54.5599, Z -7.1667, A 0.000, B 0.000, C 0.000 }
gfCNCPoint5[14807] = {X 478.4401, Y 55.2566, Z -7.1667, A 0.000, B 0.000, C 0.000 }
gfCNCPoint5[14808] = {X 478.9643, Y 56.0909, Z -7.1667, A 0.000, B 0.000, C 0.000 }
gfCNCPoint5[14809] = {X 479.2897, Y 57.0209, Z -7.1667, A 0.000, B 0.000, C 0.000 }
gfCNCPoint5[14810] = {X 479.4000, Y 58.0000, Z -7.1667, A 0.000, B 0.000, C 0.000 }
gfCNCPoint5[14811] = {X 479.3998, Y 58.9704, Z -7.1667, A 0.000, B 0.000, C 0.000 }
gfCNCPoint5[14812] = {X 479.3040, Y 59.8482, Z -7.1667, A 0.000, B 0.000, C 0.000 }
gfCNCPoint5[14813] = {X 479.0348, Y 60.6892, Z -7.1667, A 0.000, B 0.000, C 0.000 }
gfCNCPoint5[14814] = {X 478.6031, Y 61.4594, Z -7.1667, A 0.000, B 0.000, C 0.000 }
gfCNCPoint5[14815] = {X 478.0263, Y 62.1280, Z -7.1667, A 0.000, B 0.000, C 0.000 }
gfCNCPoint5[14816] = {X 477.3276, Y 62.6680, Z -7.1667, A 0.000, B 0.000, C 0.000 }
gfCNCPoint5[14817] = {X 476.5352, Y 63.0575, Z -7.1667, A 0.000, B 0.000, C 0.000 }
gfCNCPoint5[14818] = {X 475.6810, Y 63.2810, Z -7.1667, A 0.000, B 0.000, C 0.000 }
gfCNCPoint5[14819] = {X 475.6814, Y 92.7035, Z -7.1667, A 0.000, B 0.000, C 0.000 }
gfCNCPoint5[14820] = {X 476.0458, Y 92.7968, Z -7.1667, A 0.000, B 0.000, C 0.000 }
gfCNCPoint5[14821] = {X 476.4053, Y 92.9071, Z -7.1667, A 0.000, B 0.000, C 0.000 }
gfCNCPoint5[14822] = {X 477.2341, Y 93.2829, Z -7.1667, A 0.000, B 0.000, C 0.000 }
gfCNCPoint5[14823] = {X 477.9673, Y 93.8218, Z -7.1667, A 0.000, B 0.000, C 0.000 }
gfCNCPoint5[14824] = {X 478.5733, Y 94.5007, Z -7.1667, A 0.000, B 0.000, C 0.000 }
gfCNCPoint5[14825] = {X 479.0258, Y 95.2901, Z -7.1667, A 0.000, B 0.000, C 0.000 }
gfCNCPoint5[14826] = {X 479.3054, Y 96.1561, Z -7.1667, A 0.000, B 0.000, C 0.000 }
gfCNCPoint5[14827] = {X 479.4000, Y 97.0611, Z -7.1667, A 0.000, B 0.000, C 0.000 }
gfCNCPoint5[14828] = {X 479.4000, Y 97.6951, Z -7.1667, A 0.000, B 0.000, C 0.000 }
gfCNCPoint5[14829] = {X 479.8800, Y 97.6951, Z -7.1667, A 0.000, B 0.000, C 0.000 }
gfCNCPoint5[14830] = {X 507.6812, Y 97.6951, Z -7.1667, A 0.000, B 0.000, C 0.000 }
gfCNCPoint5[14831] = {X 507.6812, Y 100.0951, Z -7.1667, A 0.000, B 0.000, C 0.000 }
gfCNCPoint5[14832] = {X 600.0147, Y 100.0951, Z -7.1667, A 0.000, B 0.000, C 0.000 }
gfCNCPoint5[14833] = {X 600.0672, Y 100.0699, Z -7.1667, A 0.000, B 0.000, C 0.000 }
gfCNCPoint5[14834] = {X 600.0950, Y 100.0186, Z -7.1667, A 0.000, B 0.000, C 0.000 }
gfCNCPoint5[14835] = {X 600.0967, Y 99.1432, Z -7.1667, A 0.000, B 0.000, C 0.000 }
gfCNCPoint5[14836] = {X 600.0967, Y 49.8790, Z -7.1667, A 0.000, B 0.000, C 0.000 }
gfCNCPoint5[14837] = {X 601.1113, Y 49.7518, Z -7.1667, A 0.000, B 0.000, C 0.000 }
gfCNCPoint5[14838] = {X 602.0771, Y 49.4159, Z -7.1667, A 0.000, B 0.000, C 0.000 }
gfCNCPoint5[14839] = {X 602.9517, Y 48.8861, Z -7.1667, A 0.000, B 0.000, C 0.000 }
gfCNCPoint5[14840] = {X 603.6967, Y 48.1858, Z -7.1667, A 0.000, B 0.000, C 0.000 }
gfCNCPoint5[14841] = {X 603.6967, Y 47.3863, Z -7.1667, A 0.000, B 0.000, C 0.000 }
gfCNCPoint5[14842] = {X 603.1504, Y 48.0717, Z -7.1667, A 0.000, B 0.000, C 0.000 }
gfCNCPoint5[14843] = {X 602.4791, Y 48.6351, Z -7.1667, A 0.000, B 0.000, C 0.000 }
gfCNCPoint5[14844] = {X 601.7095, Y 49.0543, Z -7.1667, A 0.000, B 0.000, C 0.000 }
gfCNCPoint5[14845] = {X 600.8720, Y 49.3127, Z -7.1667, A 0.000, B 0.000, C 0.000 }
gfCNCPoint5[14846] = {X 600.0000, Y 49.4000, Z -7.1667, A 0.000, B 0.000, C 0.000 }
gfCNCPoint5[14847] = {X 593.5565, Y 49.4000, Z -7.1667, A 0.000, B 0.000, C 0.000 }
gfCNCPoint5[14848] = {X 592.5988, Y 49.2945, Z -7.1667, A 0.000, B 0.000, C 0.000 }
gfCNCPoint5[14849] = {X 591.6870, Y 48.9831, Z -7.1667, A 0.000, B 0.000, C 0.000 }
gfCNCPoint5[14850] = {X 590.8648, Y 48.4806, Z -7.1667, A 0.000, B 0.000, C 0.000 }
gfCNCPoint5[14851] = {X 590.1717, Y 47.8112, Z -7.1667, A 0.000, B 0.000, C 0.000 }
gfCNCPoint5[14852] = {X 589.6410, Y 47.0071, Z -7.1667, A 0.000, B 0.000, C 0.000 }
gfCNCPoint5[14853] = {X 589.3741, Y 46.3664, Z -7.1667, A 0.000, B 0.000, C 0.000 }
gfCNCPoint5[14854] = {X 589.2113, Y 45.6918, Z -7.1667, A 0.000, B 0.000, C 0.000 }
gfCNCPoint5[14855] = {X 589.1565, Y 45.0000, Z -7.1667, A 0.000, B 0.000, C 0.000 }
gfCNCPoint5[14856] = {X 589.1565, Y 44.0644, Z -7.1667, A 0.000, B 0.000, C 0.000 }
gfCNCPoint5[14857] = {X 589.2602, Y 43.1280, Z -7.1667, A 0.000, B 0.000, C 0.000 }
gfCNCPoint5[14858] = {X 589.5593, Y 42.2347, Z -7.1667, A 0.000, B 0.000, C 0.000 }
gfCNCPoint5[14859] = {X 590.0401, Y 41.4246, Z -7.1667, A 0.000, B 0.000, C 0.000 }
gfCNCPoint5[14860] = {X 590.6812, Y 40.7342, Z -7.1667, A 0.000, B 0.000, C 0.000 }
gfCNCPoint5[14861] = {X 590.6819, Y 33.9435, Z -7.1667, A 0.000, B 0.000, C 0.000 }
gfCNCPoint5[14862] = {X 585.5192, Y 46.6830, Z -7.1667, A 0.000, B 0.000, C 0.000 }
gfCNCPoint5[14863] = {X 585.4476, Y 46.8466, Z -7.1667, A 0.000, B 0.000, C 0.000 }
gfCNCPoint5[14864] = {X 585.3694, Y 47.0071, Z -7.1667, A 0.000, B 0.000, C 0.000 }
gfCNCPoint5[14865] = {X 584.8417, Y 47.8075, Z -7.1667, A 0.000, B 0.000, C 0.000 }
gfCNCPoint5[14866] = {X 584.1532, Y 48.4747, Z -7.1667, A 0.000, B 0.000, C 0.000 }
gfCNCPoint5[14867] = {X 583.3365, Y 48.9769, Z -7.1667, A 0.000, B 0.000, C 0.000 }
gfCNCPoint5[14868] = {X 582.4111, Y 49.2946, Z -7.1667, A 0.000, B 0.000, C 0.000 }
gfCNCPoint5[14869] = {X 581.4384, Y 49.4000, Z -7.1667, A 0.000, B 0.000, C 0.000 }
gfCNCPoint5[14870] = {X 580.4664, Y 49.2878, Z -7.1667, A 0.000, B 0.000, C 0.000 }
gfCNCPoint5[14871] = {X 579.5433, Y 48.9635, Z -7.1667, A 0.000, B 0.000, C 0.000 }
gfCNCPoint5[14872] = {X 578.7146, Y 48.4433, Z -7.1667, A 0.000, B 0.000, C 0.000 }
gfCNCPoint5[14873] = {X 578.0214, Y 47.7529, Z -7.1667, A 0.000, B 0.000, C 0.000 }
gfCNCPoint5[14874] = {X 577.4979, Y 46.9263, Z -7.1667, A 0.000, B 0.000, C 0.000 }
gfCNCPoint5[14875] = {X 577.4375, Y 46.7968, Z -7.1667, A 0.000, B 0.000, C 0.000 }
gfCNCPoint5[14876] = {X 577.3813, Y 46.6655, Z -7.1667, A 0.000, B 0.000, C 0.000 }
gfCNCPoint5[14877] = {X 572.0999, Y 33.7510, Z -7.1667, A 0.000, B 0.000, C 0.000 }
gfCNCPoint5[14878] = {X 572.1001, Y 40.7340, Z -7.1667, A 0.000, B 0.000, C 0.000 }
gfCNCPoint5[14879] = {X 572.7442, Y 41.4230, Z -7.1667, A 0.000, B 0.000, C 0.000 }
gfCNCPoint5[14880] = {X 573.2267, Y 42.2335, Z -7.1667, A 0.000, B 0.000, C 0.000 }
gfCNCPoint5[14881] = {X 573.5253, Y 43.1282, Z -7.1667, A 0.000, B 0.000, C 0.000 }
gfCNCPoint5[14882] = {X 573.6264, Y 44.0660, Z -7.1667, A 0.000, B 0.000, C 0.000 }
gfCNCPoint5[14883] = {X 573.6264, Y 45.0000, Z -7.1667, A 0.000, B 0.000, C 0.000 }
gfCNCPoint5[14884] = {X 573.5140, Y 45.9884, Z -7.1667, A 0.000, B 0.000, C 0.000 }
gfCNCPoint5[14885] = {X 573.1824, Y 46.9263, Z -7.1667, A 0.000, B 0.000, C 0.000 }
gfCNCPoint5[14886] = {X 572.6569, Y 47.7553, Z -7.1667, A 0.000, B 0.000, C 0.000 }
gfCNCPoint5[14887] = {X 571.9608, Y 48.4472, Z -7.1667, A 0.000, B 0.000, C 0.000 }
gfCNCPoint5[14888] = {X 571.1286, Y 48.9676, Z -7.1667, A 0.000, B 0.000, C 0.000 }
gfCNCPoint5[14889] = {X 570.2018, Y 49.2905, Z -7.1667, A 0.000, B 0.000, C 0.000 }
gfCNCPoint5[14890] = {X 569.2264, Y 49.4000, Z -7.1667, A 0.000, B 0.000, C 0.000 }
gfCNCPoint5[14891] = {X 562.4443, Y 49.4000, Z -7.1667, A 0.000, B 0.000, C 0.000 }
gfCNCPoint5[14892] = {X 561.5859, Y 49.3155, Z -7.1667, A 0.000, B 0.000, C 0.000 }
gfCNCPoint5[14893] = {X 560.7605, Y 49.0651, Z -7.1667, A 0.000, B 0.000, C 0.000 }
gfCNCPoint5[14894] = {X 559.9998, Y 48.6585, Z -7.1667, A 0.000, B 0.000, C 0.000 }
gfCNCPoint5[14895] = {X 559.3330, Y 48.1113, Z -7.1667, A 0.000, B 0.000, C 0.000 }
gfCNCPoint5[14896] = {X 558.7858, Y 47.4445, Z -7.1667, A 0.000, B 0.000, C 0.000 }
gfCNCPoint5[14897] = {X 558.3792, Y 46.6838, Z -7.1667, A 0.000, B 0.000, C 0.000 }
gfCNCPoint5[14898] = {X 558.1288, Y 45.8584, Z -7.1667, A 0.000, B 0.000, C 0.000 }
gfCNCPoint5[14899] = {X 558.0443, Y 45.0000, Z -7.1667, A 0.000, B 0.000, C 0.000 }
gfCNCPoint5[14900] = {X 558.0443, Y 44.0646, Z -7.1667, A 0.000, B 0.000, C 0.000 }
gfCNCPoint5[14901] = {X 558.1477, Y 43.1277, Z -7.1667, A 0.000, B 0.000, C 0.000 }
gfCNCPoint5[14902] = {X 558.4471, Y 42.2339, Z -7.1667, A 0.000, B 0.000, C 0.000 }
gfCNCPoint5[14903] = {X 558.9287, Y 41.4237, Z -7.1667, A 0.000, B 0.000, C 0.000 }
gfCNCPoint5[14904] = {X 559.5709, Y 40.7337, Z -7.1667, A 0.000, B 0.000, C 0.000 }
gfCNCPoint5[14905] = {X 559.5710, Y 9.2664, Z -7.1667, A 0.000, B 0.000, C 0.000 }
gfCNCPoint5[14906] = {X 558.9267, Y 8.5773, Z -7.1667, A 0.000, B 0.000, C 0.000 }
gfCNCPoint5[14907] = {X 558.4441, Y 7.7667, Z -7.1667, A 0.000, B 0.000, C 0.000 }
gfCNCPoint5[14908] = {X 558.1454, Y 6.8719, Z -7.1667, A 0.000, B 0.000, C 0.000 }
gfCNCPoint5[14909] = {X 558.0443, Y 5.9340, Z -7.1667, A 0.000, B 0.000, C 0.000 }
gfCNCPoint5[14910] = {X 558.0443, Y 5.0000, Z -7.1667, A 0.000, B 0.000, C 0.000 }
gfCNCPoint5[14911] = {X 558.1353, Y 4.1096, Z -7.1667, A 0.000, B 0.000, C 0.000 }
gfCNCPoint5[14912] = {X 558.4046, Y 3.2561, Z -7.1667, A 0.000, B 0.000, C 0.000 }
gfCNCPoint5[14913] = {X 558.9156, Y 2.3717, Z -7.1667, A 0.000, B 0.000, C 0.000 }
gfCNCPoint5[14914] = {X 559.6166, Y 1.6289, Z -7.1667, A 0.000, B 0.000, C 0.000 }
gfCNCPoint5[14915] = {X 560.4700, Y 1.0678, Z -7.1667, A 0.000, B 0.000, C 0.000 }
gfCNCPoint5[14916] = {X 561.4298, Y 0.7185, Z -7.1667, A 0.000, B 0.000, C 0.000 }
gfCNCPoint5[14917] = {X 562.4443, Y 0.6000, Z -7.1667, A 0.000, B 0.000, C 0.000 }
gfCNCPoint5[14918] = {X 570.9376, Y 0.6000, Z -7.1667, A 0.000, B 0.000, C 0.000 }
gfCNCPoint5[14919] = {X 571.9520, Y 0.7185, Z -7.1667, A 0.000, B 0.000, C 0.000 }
gfCNCPoint5[14920] = {X 572.9118, Y 1.0678, Z -7.1667, A 0.000, B 0.000, C 0.000 }
gfCNCPoint5[14921] = {X 573.7652, Y 1.6289, Z -7.1667, A 0.000, B 0.000, C 0.000 }
gfCNCPoint5[14922] = {X 574.4663, Y 2.3717, Z -7.1667, A 0.000, B 0.000, C 0.000 }
gfCNCPoint5[14923] = {X 574.9772, Y 3.2561, Z -7.1667, A 0.000, B 0.000, C 0.000 }
gfCNCPoint5[14924] = {X 575.2465, Y 4.1096, Z -7.1667, A 0.000, B 0.000, C 0.000 }
gfCNCPoint5[14925] = {X 575.3376, Y 5.0000, Z -7.1667, A 0.000, B 0.000, C 0.000 }
gfCNCPoint5[14926] = {X 575.3372, Y 5.9910, Z -7.1667, A 0.000, B 0.000, C 0.000 }
gfCNCPoint5[14927] = {X 575.2577, Y 6.7683, Z -7.1667, A 0.000, B 0.000, C 0.000 }
gfCNCPoint5[14928] = {X 575.0420, Y 7.5194, Z -7.1667, A 0.000, B 0.000, C 0.000 }
gfCNCPoint5[14929] = {X 574.6969, Y 8.2205, Z -7.1667, A 0.000, B 0.000, C 0.000 }
gfCNCPoint5[14930] = {X 575.2866, Y 9.6559, Z -7.1667, A 0.000, B 0.000, C 0.000 }
gfCNCPoint5[14931] = {X 580.9325, Y 23.5214, Z -7.1667, A 0.000, B 0.000, C 0.000 }
gfCNCPoint5[14932] = {X 581.1912, Y 24.1568, Z -7.1667, A 0.000, B 0.000, C 0.000 }
gfCNCPoint5[14933] = {X 587.7567, Y 8.0995, Z -7.1667, A 0.000, B 0.000, C 0.000 }
gfCNCPoint5[14934] = {X 587.4433, Y 7.4140, Z -7.1667, A 0.000, B 0.000, C 0.000 }
gfCNCPoint5[14935] = {X 587.2515, Y 6.6850, Z -7.1667, A 0.000, B 0.000, C 0.000 }
gfCNCPoint5[14936] = {X 587.1870, Y 5.9340, Z -7.1667, A 0.000, B 0.000, C 0.000 }
gfCNCPoint5[14937] = {X 587.1870, Y 5.0000, Z -7.1667, A 0.000, B 0.000, C 0.000 }
gfCNCPoint5[14938] = {X 587.2780, Y 4.1096, Z -7.1667, A 0.000, B 0.000, C 0.000 }
gfCNCPoint5[14939] = {X 587.5473, Y 3.2561, Z -7.1667, A 0.000, B 0.000, C 0.000 }
gfCNCPoint5[14940] = {X 587.7249, Y 2.8918, Z -7.1667, A 0.000, B 0.000, C 0.000 }
gfCNCPoint5[14941] = {X 587.9353, Y 2.5453, Z -7.1667, A 0.000, B 0.000, C 0.000 }
gfCNCPoint5[14942] = {X 588.4826, Y 1.8818, Z -7.1667, A 0.000, B 0.000, C 0.000 }
gfCNCPoint5[14943] = {X 589.1485, Y 1.3375, Z -7.1667, A 0.000, B 0.000, C 0.000 }
gfCNCPoint5[14944] = {X 589.9077, Y 0.9331, Z -7.1667, A 0.000, B 0.000, C 0.000 }
gfCNCPoint5[14945] = {X 590.7310, Y 0.6841, Z -7.1667, A 0.000, B 0.000, C 0.000 }
gfCNCPoint5[14946] = {X 591.5870, Y 0.6000, Z -7.1667, A 0.000, B 0.000, C 0.000 }
gfCNCPoint5[14947] = {X 600.0000, Y 0.6000, Z -7.1667, A 0.000, B 0.000, C 0.000 }
gfCNCPoint5[14948] = {X 600.8720, Y 0.6873, Z -7.1667, A 0.000, B 0.000, C 0.000 }
gfCNCPoint5[14949] = {X 601.7095, Y 0.9457, Z -7.1667, A 0.000, B 0.000, C 0.000 }
gfCNCPoint5[14950] = {X 602.4791, Y 1.3649, Z -7.1667, A 0.000, B 0.000, C 0.000 }
gfCNCPoint5[14951] = {X 603.1504, Y 1.9283, Z -7.1667, A 0.000, B 0.000, C 0.000 }
gfCNCPoint5[14952] = {X 603.6967, Y 2.6137, Z -7.1667, A 0.000, B 0.000, C 0.000 }
gfCNCPoint5[14953] = {X 603.6967, Y 1.8142, Z -7.1667, A 0.000, B 0.000, C 0.000 }
gfCNCPoint5[14954] = {X 602.9514, Y 1.1136, Z -7.1667, A 0.000, B 0.000, C 0.000 }
gfCNCPoint5[14955] = {X 602.0764, Y 0.5838, Z -7.1667, A 0.000, B 0.000, C 0.000 }
gfCNCPoint5[14956] = {X 601.1102, Y 0.2480, Z -7.1667, A 0.000, B 0.000, C 0.000 }
gfCNCPoint5[14957] = {X 600.0952, Y 0.1209, Z -7.1667, A 0.000, B 0.000, C 0.000 }
gfCNCPoint5[14958] = {X 600.0950, Y -0.0186, Z -7.1667, A 0.000, B 0.000, C 0.000 }
gfCNCPoint5[14959] = {X 600.0672, Y -0.0699, Z -7.1667, A 0.000, B 0.000, C 0.000 }
gfCNCPoint5[14960] = {X 600.0147, Y -0.0951, Z -7.1667, A 0.000, B 0.000, C 0.000 }
gfCNCPoint5[14961] = {X 580.1328, Y -0.0951, Z -7.1667, A 0.000, B 0.000, C 0.000 }
gfCNCPoint5[14962] = {X 580.1328, Y 4.7049, Z -7.1667, A 0.000, B 0.000, C 0.000 }
gfCNCPoint5[14963] = {X 580.1364, Y 4.8524, Z -7.1667, A 0.000, B 0.000, C 0.000 }
gfCNCPoint5[14964] = {X 580.1376, Y 5.0000, Z -7.1667, A 0.000, B 0.000, C 0.000 }
gfCNCPoint5[14965] = {X 580.1376, Y 5.9339, Z -7.1667, A 0.000, B 0.000, C 0.000 }
gfCNCPoint5[14966] = {X 580.0684, Y 7.0597, Z -7.1667, A 0.000, B 0.000, C 0.000 }
gfCNCPoint5[14967] = {X 579.8621, Y 8.1685, Z -7.1667, A 0.000, B 0.000, C 0.000 }
gfCNCPoint5[14968] = {X 581.1999, Y 11.4527, Z -7.1667, A 0.000, B 0.000, C 0.000 }
gfCNCPoint5[14969] = {X 582.6182, Y 7.9840, Z -7.1667, A 0.000, B 0.000, C 0.000 }
gfCNCPoint5[14970] = {X 582.4488, Y 6.9992, Z -7.1667, A 0.000, B 0.000, C 0.000 }
gfCNCPoint5[14971] = {X 582.3872, Y 6.0018, Z -7.1667, A 0.000, B 0.000, C 0.000 }
gfCNCPoint5[14972] = {X 582.3870, Y 5.0000, Z -7.1667, A 0.000, B 0.000, C 0.000 }
gfCNCPoint5[14973] = {X 582.3881, Y 4.8524, Z -7.1667, A 0.000, B 0.000, C 0.000 }
gfCNCPoint5[14974] = {X 582.3917, Y 4.7049, Z -7.1667, A 0.000, B 0.000, C 0.000 }
gfCNCPoint5[14975] = {X 580.1328, Y 4.7049, Z -7.1667, A 0.000, B 0.000, C 0.000 }
gfCNCPoint5[14976] = {X 580.1328, Y 2.3049, Z -7.1667, A 0.000, B 0.000, C 0.000 }
gfCNCPoint5[14977] = {X 577.1807, Y 2.3049, Z -7.1667, A 0.000, B 0.000, C 0.000 }
gfCNCPoint5[14978] = {X 577.5739, Y 3.5173, Z -7.1667, A 0.000, B 0.000, C 0.000 }
gfCNCPoint5[14979] = {X 577.7341, Y 4.7819, Z -7.1667, A 0.000, B 0.000, C 0.000 }
gfCNCPoint5[14980] = {X 577.7367, Y 4.8909, Z -7.1667, A 0.000, B 0.000, C 0.000 }
gfCNCPoint5[14981] = {X 577.7376, Y 5.0000, Z -7.1667, A 0.000, B 0.000, C 0.000 }
gfCNCPoint5[14982] = {X 577.7376, Y 5.9339, Z -7.1667, A 0.000, B 0.000, C 0.000 }
gfCNCPoint5[14983] = {X 577.6319, Y 7.1282, Z -7.1667, A 0.000, B 0.000, C 0.000 }
gfCNCPoint5[14984] = {X 577.3181, Y 8.2853, Z -7.1667, A 0.000, B 0.000, C 0.000 }
gfCNCPoint5[14985] = {X 581.1958, Y 17.8042, Z -7.1667, A 0.000, B 0.000, C 0.000 }
gfCNCPoint5[14986] = {X 585.1513, Y 8.1301, Z -7.1667, A 0.000, B 0.000, C 0.000 }
gfCNCPoint5[14987] = {X 584.8834, Y 7.0754, Z -7.1667, A 0.000, B 0.000, C 0.000 }
gfCNCPoint5[14988] = {X 584.7872, Y 5.9914, Z -7.1667, A 0.000, B 0.000, C 0.000 }
gfCNCPoint5[14989] = {X 584.7870, Y 5.0000, Z -7.1667, A 0.000, B 0.000, C 0.000 }
gfCNCPoint5[14990] = {X 584.7878, Y 4.8909, Z -7.1667, A 0.000, B 0.000, C 0.000 }
gfCNCPoint5[14991] = {X 584.7905, Y 4.7819, Z -7.1667, A 0.000, B 0.000, C 0.000 }
gfCNCPoint5[14992] = {X 584.9506, Y 3.5173, Z -7.1667, A 0.000, B 0.000, C 0.000 }
gfCNCPoint5[14993] = {X 585.3439, Y 2.3049, Z -7.1667, A 0.000, B 0.000, C 0.000 }
gfCNCPoint5[14994] = {X 580.1328, Y 2.3049, Z -7.1667, A 0.000, B 0.000, C 0.000 }
gfCNCPoint5[14995] = {X 580.1328, Y -0.0951, Z -7.1667, A 0.000, B 0.000, C 0.000 }
gfCNCPoint5[14996] = {X 351.5697, Y -0.0951, Z -7.1667, A 0.000, B 0.000, C 0.000 }
gfCNCPoint5[14997] = {X 351.4403, Y -0.1194, Z -7.1667, A 0.000, B 0.000, C 0.000 }
gfCNCPoint5[14998] = {X 348.9371, Y -0.4688, Z -7.1667, A 0.000, B 0.000, C 0.000 }
gfCNCPoint5[14999] = {X 346.4122, Y -0.5816, Z -7.1667, A 0.000, B 0.000, C 0.000 }
gfCNCPoint5[15000] = {X 343.8878, Y -0.4566, Z -7.1667, A 0.000, B 0.000, C 0.000 }
gfCNCPoint5[15001] = {X 341.3863, Y -0.0951, Z -7.1667, A 0.000, B 0.000, C 0.000 }
gfCNCPoint5[15002] = {X -0.0147, Y -0.0951, Z -7.1667, A 0.000, B 0.000, C 0.000 }
gfCNCPoint5[15003] = {X -0.0672, Y -0.0699, Z -7.1667, A 0.000, B 0.000, C 0.000 }
gfCNCPoint5[15004] = {X -0.0950, Y -0.0186, Z -7.1667, A 0.000, B 0.000, C 0.000 }
gfCNCPoint5[15005] = {X -0.0967, Y 0.8568, Z -7.1667, A 0.000, B 0.000, C 0.000 }
gfCNCPoint5[15006] = {X -0.0967, Y 8.7891, Z -7.1667, A 0.000, B 0.000, C 0.000 }
gfCNCPoint5[15007] = {X -0.7634, Y 8.9979, Z -7.1667, A 0.000, B 0.000, C 0.000 }
gfCNCPoint5[15008] = {X -1.3934, Y 9.2998, Z -7.1667, A 0.000, B 0.000, C 0.000 }
gfCNCPoint5[15009] = {X -1.9904, Y 9.6404, Z -7.1667, A 0.000, B 0.000, C 0.000 }
gfCNCPoint5[15010] = {X -2.6455, Y 10.0885, Z -7.1667, A 0.000, B 0.000, C 0.000 }
gfCNCPoint5[15011] = {X -3.2193, Y 10.6367, Z -7.1667, A 0.000, B 0.000, C 0.000 }
gfCNCPoint5[15012] = {X -3.6967, Y 11.2708, Z -7.1667, A 0.000, B 0.000, C 0.000 }
gfCNCPoint5[15013] = {X -3.6967, Y 12.3465, Z -7.1667, A 0.000, B 0.000, C 0.000 }
gfCNCPoint5[15014] = {X -3.2333, Y 11.4386, Z -7.1667, A 0.000, B 0.000, C 0.000 }
gfCNCPoint5[15015] = {X -2.5735, Y 10.6616, Z -7.1667, A 0.000, B 0.000, C 0.000 }
gfCNCPoint5[15016] = {X -1.7526, Y 10.0573, Z -7.1667, A 0.000, B 0.000, C 0.000 }
gfCNCPoint5[15017] = {X -1.0994, Y 9.6852, Z -7.1667, A 0.000, B 0.000, C 0.000 }
gfCNCPoint5[15018] = {X -0.1608, Y 9.3012, Z -7.1667, A 0.000, B 0.000, C 0.000 }
gfCNCPoint5[15019] = {X 0.8408, Y 9.1423, Z -7.1667, A 0.000, B 0.000, C 0.000 }
gfCNCPoint5[15020] = {X 1.8521, Y 9.2169, Z -7.1667, A 0.000, B 0.000, C 0.000 }
gfCNCPoint5[15021] = {X 2.2303, Y 9.3068, Z -7.1667, A 0.000, B 0.000, C 0.000 }
gfCNCPoint5[15022] = {X 2.5991, Y 9.4297, Z -7.1667, A 0.000, B 0.000, C 0.000 }
gfCNCPoint5[15023] = {X 3.4586, Y 9.0453, Z -7.1667, A 0.000, B 0.000, C 0.000 }
gfCNCPoint5[15024] = {X 5.5423, Y 8.2603, Z -7.1667, A 0.000, B 0.000, C 0.000 }
gfCNCPoint5[15025] = {X 7.6901, Y 7.6728, Z -7.1667, A 0.000, B 0.000, C 0.000 }
gfCNCPoint5[15026] = {X 9.8832, Y 7.2879, Z -7.1667, A 0.000, B 0.000, C 0.000 }
gfCNCPoint5[15027] = {X 12.1027, Y 7.1089, Z -7.1667, A 0.000, B 0.000, C 0.000 }
gfCNCPoint5[15028] = {X 14.3292, Y 7.1374, Z -7.1667, A 0.000, B 0.000, C 0.000 }
gfCNCPoint5[15029] = {X 16.5434, Y 7.3732, Z -7.1667, A 0.000, B 0.000, C 0.000 }
gfCNCPoint5[15030] = {X 18.2870, Y 7.7303, Z -7.1667, A 0.000, B 0.000, C 0.000 }
gfCNCPoint5[15031] = {X 19.9854, Y 8.2624, Z -7.1667, A 0.000, B 0.000, C 0.000 }
gfCNCPoint5[15032] = {X 21.6211, Y 8.9640, Z -7.1667, A 0.000, B 0.000, C 0.000 }
gfCNCPoint5[15033] = {X 23.1772, Y 9.8278, Z -7.1667, A 0.000, B 0.000, C 0.000 }
gfCNCPoint5[15034] = {X 24.6376, Y 10.8451, Z -7.1667, A 0.000, B 0.000, C 0.000 }
gfCNCPoint5[15035] = {X 25.7302, Y 11.8007, Z -7.1667, A 0.000, B 0.000, C 0.000 }
gfCNCPoint5[15036] = {X 26.7103, Y 12.8714, Z -7.1667, A 0.000, B 0.000, C 0.000 }
gfCNCPoint5[15037] = {X 27.5657, Y 14.0442, Z -7.1667, A 0.000, B 0.000, C 0.000 }
gfCNCPoint5[15038] = {X 28.2859, Y 15.3044, Z -7.1667, A 0.000, B 0.000, C 0.000 }
gfCNCPoint5[15039] = {X 28.8621, Y 16.6367, Z -7.1667, A 0.000, B 0.000, C 0.000 }
gfCNCPoint5[15040] = {X 29.3387, Y 18.3012, Z -7.1667, A 0.000, B 0.000, C 0.000 }
gfCNCPoint5[15041] = {X 29.6216, Y 20.0094, Z -7.1667, A 0.000, B 0.000, C 0.000 }
gfCNCPoint5[15042] = {X 29.7068, Y 21.7387, Z -7.1667, A 0.000, B 0.000, C 0.000 }
gfCNCPoint5[15043] = {X 29.5932, Y 23.4664, Z -7.1667, A 0.000, B 0.000, C 0.000 }
gfCNCPoint5[15044] = {X 29.2825, Y 25.1697, Z -7.1667, A 0.000, B 0.000, C 0.000 }
gfCNCPoint5[15045] = {X 28.7909, Y 26.7456, Z -7.1667, A 0.000, B 0.000, C 0.000 }
gfCNCPoint5[15046] = {X 28.0838, Y 28.2372, Z -7.1667, A 0.000, B 0.000, C 0.000 }
gfCNCPoint5[15047] = {X 27.1750, Y 29.6153, Z -7.1667, A 0.000, B 0.000, C 0.000 }
gfCNCPoint5[15048] = {X 26.3579, Y 30.5724, Z -7.1667, A 0.000, B 0.000, C 0.000 }
gfCNCPoint5[15049] = {X 25.4434, Y 31.4368, Z -7.1667, A 0.000, B 0.000, C 0.000 }
gfCNCPoint5[15050] = {X 25.6940, Y 31.5324, Z -7.1667, A 0.000, B 0.000, C 0.000 }
gfCNCPoint5[15051] = {X 25.9383, Y 31.6432, Z -7.1667, A 0.000, B 0.000, C 0.000 }
gfCNCPoint5[15052] = {X 26.5119, Y 31.9806, Z -7.1667, A 0.000, B 0.000, C 0.000 }
gfCNCPoint5[15053] = {X 27.0280, Y 32.4007, Z -7.1667, A 0.000, B 0.000, C 0.000 }
gfCNCPoint5[15054] = {X 27.1608, Y 32.5321, Z -7.1667, A 0.000, B 0.000, C 0.000 }
gfCNCPoint5[15055] = {X 27.2878, Y 32.6689, Z -7.1667, A 0.000, B 0.000, C 0.000 }
gfCNCPoint5[15056] = {X 27.6592, Y 33.1494, Z -7.1667, A 0.000, B 0.000, C 0.000 }
gfCNCPoint5[15057] = {X 27.9608, Y 33.6765, Z -7.1667, A 0.000, B 0.000, C 0.000 }
gfCNCPoint5[15058] = {X 30.9820, Y 39.9182, Z -7.1667, A 0.000, B 0.000, C 0.000 }
gfCNCPoint5[15059] = {X 31.3085, Y 40.8441, Z -7.1667, A 0.000, B 0.000, C 0.000 }
gfCNCPoint5[15060] = {X 31.4215, Y 41.8194, Z -7.1667, A 0.000, B 0.000, C 0.000 }
gfCNCPoint5[15061] = {X 31.3155, Y 42.7955, Z -7.1667, A 0.000, B 0.000, C 0.000 }
gfCNCPoint5[15062] = {X 30.9956, Y 43.7238, Z -7.1667, A 0.000, B 0.000, C 0.000 }
gfCNCPoint5[15063] = {X 30.4779, Y 44.5580, Z -7.1667, A 0.000, B 0.000, C 0.000 }
gfCNCPoint5[15064] = {X 29.7880, Y 45.2567, Z -7.1667, A 0.000, B 0.000, C 0.000 }
gfCNCPoint5[15065] = {X 29.2521, Y 45.6900, Z -7.1667, A 0.000, B 0.000, C 0.000 }
gfCNCPoint5[15066] = {X 28.5414, Y 46.1592, Z -7.1667, A 0.000, B 0.000, C 0.000 }
gfCNCPoint5[15067] = {X 27.7538, Y 46.4830, Z -7.1667, A 0.000, B 0.000, C 0.000 }
gfCNCPoint5[15068] = {X 26.9187, Y 46.6494, Z -7.1667, A 0.000, B 0.000, C 0.000 }
gfCNCPoint5[15069] = {X 26.0672, Y 46.6523, Z -7.1667, A 0.000, B 0.000, C 0.000 }
gfCNCPoint5[15070] = {X 25.2310, Y 46.4914, Z -7.1667, A 0.000, B 0.000, C 0.000 }
gfCNCPoint5[15071] = {X 23.4348, Y 47.4371, Z -7.1667, A 0.000, B 0.000, C 0.000 }
gfCNCPoint5[15072] = {X 21.5774, Y 48.2561, Z -7.1667, A 0.000, B 0.000, C 0.000 }
gfCNCPoint5[15073] = {X 19.6678, Y 48.9445, Z -7.1667, A 0.000, B 0.000, C 0.000 }
gfCNCPoint5[15074] = {X 19.5111, Y 48.9960, Z -7.1667, A 0.000, B 0.000, C 0.000 }
gfCNCPoint5[15075] = {X 17.5875, Y 49.5251, Z -7.1667, A 0.000, B 0.000, C 0.000 }
gfCNCPoint5[15076] = {X 15.6250, Y 49.8843, Z -7.1667, A 0.000, B 0.000, C 0.000 }
gfCNCPoint5[15077] = {X 13.6386, Y 50.0708, Z -7.1667, A 0.000, B 0.000, C 0.000 }
gfCNCPoint5[15078] = {X 11.6436, Y 50.0833, Z -7.1667, A 0.000, B 0.000, C 0.000 }
gfCNCPoint5[15079] = {X 9.6551, Y 49.9216, Z -7.1667, A 0.000, B 0.000, C 0.000 }
gfCNCPoint5[15080] = {X 7.6883, Y 49.5869, Z -7.1667, A 0.000, B 0.000, C 0.000 }
gfCNCPoint5[15081] = {X 6.2182, Y 49.2058, Z -7.1667, A 0.000, B 0.000, C 0.000 }
gfCNCPoint5[15082] = {X 4.7886, Y 48.6935, Z -7.1667, A 0.000, B 0.000, C 0.000 }
gfCNCPoint5[15083] = {X 3.4111, Y 48.0541, Z -7.1667, A 0.000, B 0.000, C 0.000 }
gfCNCPoint5[15084] = {X 1.9574, Y 47.2025, Z -7.1667, A 0.000, B 0.000, C 0.000 }
gfCNCPoint5[15085] = {X 0.5963, Y 46.2095, Z -7.1667, A 0.000, B 0.000, C 0.000 }
gfCNCPoint5[15086] = {X -0.5426, Y 45.1854, Z -7.1667, A 0.000, B 0.000, C 0.000 }
gfCNCPoint5[15087] = {X -1.5542, Y 44.0354, Z -7.1667, A 0.000, B 0.000, C 0.000 }
gfCNCPoint5[15088] = {X -2.4247, Y 42.7752, Z -7.1667, A 0.000, B 0.000, C 0.000 }
gfCNCPoint5[15089] = {X -3.1421, Y 41.4220, Z -7.1667, A 0.000, B 0.000, C 0.000 }
gfCNCPoint5[15090] = {X -3.6967, Y 39.9943, Z -7.1667, A 0.000, B 0.000, C 0.000 }
gfCNCPoint5[15091] = {X -3.6967, Y 41.3560, Z -7.1667, A 0.000, B 0.000, C 0.000 }
gfCNCPoint5[15092] = {X -3.0107, Y 42.7266, Z -7.1667, A 0.000, B 0.000, C 0.000 }
gfCNCPoint5[15093] = {X -2.1746, Y 44.0111, Z -7.1667, A 0.000, B 0.000, C 0.000 }
gfCNCPoint5[15094] = {X -1.1991, Y 45.1933, Z -7.1667, A 0.000, B 0.000, C 0.000 }
gfCNCPoint5[15095] = {X -0.0967, Y 46.2581, Z -7.1667, A 0.000, B 0.000, C 0.000 }
gfCNCPoint5[15096] = {X -0.0967, Y 99.1432, Z -7.1667, A 0.000, B 0.000, C 0.000 }
gfCNCPoint5[15097] = {X -0.0950, Y 100.0186, Z -7.1667, A 0.000, B 0.000, C 0.000 }
gfCNCPoint5[15098] = {X -0.0672, Y 100.0699, Z -7.1667, A 0.000, B 0.000, C 0.000 }
gfCNCPoint5[15099] = {X -0.0147, Y 100.0951, Z -7.1667, A 0.000, B 0.000, C 0.000 }
gfCNCPoint5[15100] = {X 120.5926, Y 100.0951, Z -7.1667, A 0.000, B 0.000, C 0.000 }
gfCNCPoint5[15101] = {X 121.0614, Y 100.8813, Z -7.1667, A 0.000, B 0.000, C 0.000 }
gfCNCPoint5[15102] = {X 121.6687, Y 101.5661, Z -7.1667, A 0.000, B 0.000, C 0.000 }
gfCNCPoint5[15103] = {X 122.3933, Y 102.1254, Z -7.1667, A 0.000, B 0.000, C 0.000 }
gfCNCPoint5[15104] = {X 123.2095, Y 102.5397, Z -7.1667, A 0.000, B 0.000, C 0.000 }
gfCNCPoint5[15105] = {X 124.0887, Y 102.7942, Z -7.1667, A 0.000, B 0.000, C 0.000 }
gfCNCPoint5[15106] = {X 125.0000, Y 102.8800, Z -7.1667, A 0.000, B 0.000, C 0.000 }
gfCNCPoint5[15107] = {X 143.7791, Y 102.8800, Z -7.1667, A 0.000, B 0.000, C 0.000 }
gfCNCPoint5[15108] = {X 144.6904, Y 102.7942, Z -7.1667, A 0.000, B 0.000, C 0.000 }
gfCNCPoint5[15109] = {X 145.5696, Y 102.5397, Z -7.1667, A 0.000, B 0.000, C 0.000 }
gfCNCPoint5[15110] = {X 146.3858, Y 102.1254, Z -7.1667, A 0.000, B 0.000, C 0.000 }
gfCNCPoint5[15111] = {X 147.1104, Y 101.5661, Z -7.1667, A 0.000, B 0.000, C 0.000 }
gfCNCPoint5[15112] = {X 147.7177, Y 100.8813, Z -7.1667, A 0.000, B 0.000, C 0.000 }
gfCNCPoint5[15113] = {X 148.1865, Y 100.0951, Z -7.1667, A 0.000, B 0.000, C 0.000 }
gfCNCPoint5[15114] = {X 150.8387, Y 100.0951, Z -7.1667, A 0.000, B 0.000, C 0.000 }
gfCNCPoint5[15115] = {X 150.8387, Y 95.2951, Z -7.1667, A 0.000, B 0.000, C 0.000 }
gfCNCPoint5[15116] = {X 187.9256, Y 95.2951, Z -7.1667, A 0.000, B 0.000, C 0.000 }
gfCNCPoint5[15117] = {X 187.9777, Y 95.0991, Z -7.1667, A 0.000, B 0.000, C 0.000 }
gfCNCPoint5[15118] = {X 188.0352, Y 94.9045, Z -7.1667, A 0.000, B 0.000, C 0.000 }
gfCNCPoint5[15119] = {X 187.2619, Y 94.0602, Z -7.1667, A 0.000, B 0.000, C 0.000 }
gfCNCPoint5[15120] = {X 151.4055, Y 94.0602, Z -7.1667, A 0.000, B 0.000, C 0.000 }
gfCNCPoint5[15121] = {X 150.7066, Y 94.8345, Z -7.1667, A 0.000, B 0.000, C 0.000 }
gfCNCPoint5[15122] = {X 150.7765, Y 95.0637, Z -7.1667, A 0.000, B 0.000, C 0.000 }
gfCNCPoint5[15123] = {X 150.8387, Y 95.2951, Z -7.1667, A 0.000, B 0.000, C 0.000 }
gfCNCPoint5[15124] = {X 150.8387, Y 97.6951, Z -7.1667, A 0.000, B 0.000, C 0.000 }
gfCNCPoint5[15125] = {X 190.1070, Y 97.6951, Z -7.1667, A 0.000, B 0.000, C 0.000 }
gfCNCPoint5[15126] = {X 190.1070, Y 97.0659, Z -7.1667, A 0.000, B 0.000, C 0.000 }
gfCNCPoint5[15127] = {X 190.1938, Y 96.1495, Z -7.1667, A 0.000, B 0.000, C 0.000 }
gfCNCPoint5[15128] = {X 190.4511, Y 95.2657, Z -7.1667, A 0.000, B 0.000, C 0.000 }
gfCNCPoint5[15129] = {X 190.8699, Y 94.4460, Z -7.1667, A 0.000, B 0.000, C 0.000 }
gfCNCPoint5[15130] = {X 188.3182, Y 91.6602, Z -7.1667, A 0.000, B 0.000, C 0.000 }
gfCNCPoint5[15131] = {X 150.3387, Y 91.6602, Z -7.1667, A 0.000, B 0.000, C 0.000 }
gfCNCPoint5[15132] = {X 147.8646, Y 94.4013, Z -7.1667, A 0.000, B 0.000, C 0.000 }
gfCNCPoint5[15133] = {X 148.2991, Y 95.2323, Z -7.1667, A 0.000, B 0.000, C 0.000 }
gfCNCPoint5[15134] = {X 148.5672, Y 96.1309, Z -7.1667, A 0.000, B 0.000, C 0.000 }
gfCNCPoint5[15135] = {X 148.6591, Y 97.0641, Z -7.1667, A 0.000, B 0.000, C 0.000 }
gfCNCPoint5[15136] = {X 148.6591, Y 97.6951, Z -7.1667, A 0.000, B 0.000, C 0.000 }
gfCNCPoint5[15137] = {X 150.8387, Y 97.6951, Z -7.1667, A 0.000, B 0.000, C 0.000 }
gfCNCPoint5[15138] = {X 150.8387, Y 100.0951, Z -7.1667, A 0.000, B 0.000, C 0.000 }
gfCNCPoint5[15139] = {X 190.5796, Y 100.0951, Z -7.1667, A 0.000, B 0.000, C 0.000 }
gfCNCPoint5[15140] = {X 191.0484, Y 100.8813, Z -7.1667, A 0.000, B 0.000, C 0.000 }
gfCNCPoint5[15141] = {X 191.6557, Y 101.5661, Z -7.1667, A 0.000, B 0.000, C 0.000 }
gfCNCPoint5[15142] = {X 192.3802, Y 102.1254, Z -7.1667, A 0.000, B 0.000, C 0.000 }
gfCNCPoint5[15143] = {X 193.1965, Y 102.5397, Z -7.1667, A 0.000, B 0.000, C 0.000 }
gfCNCPoint5[15144] = {X 194.0757, Y 102.7942, Z -7.1667, A 0.000, B 0.000, C 0.000 }
gfCNCPoint5[15145] = {X 194.9870, Y 102.8800, Z -7.1667, A 0.000, B 0.000, C 0.000 }
gfCNCPoint5[15146] = {X 212.6141, Y 102.8800, Z -7.1667, A 0.000, B 0.000, C 0.000 }
gfCNCPoint5[15147] = {X 213.0066, Y 102.8642, Z -7.1667, A 0.000, B 0.000, C 0.000 }
gfCNCPoint5[15148] = {X 213.3966, Y 102.8169, Z -7.1667, A 0.000, B 0.000, C 0.000 }
gfCNCPoint5[15149] = {X 213.7865, Y 102.8642, Z -7.1667, A 0.000, B 0.000, C 0.000 }
gfCNCPoint5[15150] = {X 214.1790, Y 102.8800, Z -7.1667, A 0.000, B 0.000, C 0.000 }
gfCNCPoint5[15151] = {X 233.4798, Y 102.8800, Z -7.1667, A 0.000, B 0.000, C 0.000 }
gfCNCPoint5[15152] = {X 234.3911, Y 102.7942, Z -7.1667, A 0.000, B 0.000, C 0.000 }
gfCNCPoint5[15153] = {X 235.2703, Y 102.5397, Z -7.1667, A 0.000, B 0.000, C 0.000 }
gfCNCPoint5[15154] = {X 236.0865, Y 102.1254, Z -7.1667, A 0.000, B 0.000, C 0.000 }
gfCNCPoint5[15155] = {X 236.8110, Y 101.5661, Z -7.1667, A 0.000, B 0.000, C 0.000 }
gfCNCPoint5[15156] = {X 237.4184, Y 100.8813, Z -7.1667, A 0.000, B 0.000, C 0.000 }
gfCNCPoint5[15157] = {X 237.8871, Y 100.0951, Z -7.1667, A 0.000, B 0.000, C 0.000 }
gfCNCPoint5[15158] = {X 261.4785, Y 100.0951, Z -7.1667, A 0.000, B 0.000, C 0.000 }
gfCNCPoint5[15159] = {X 261.4785, Y 90.4951, Z -7.1667, A 0.000, B 0.000, C 0.000 }
gfCNCPoint5[15160] = {X 266.0961, Y 90.4951, Z -7.1667, A 0.000, B 0.000, C 0.000 }
gfCNCPoint5[15161] = {X 266.1751, Y 90.3748, Z -7.1667, A 0.000, B 0.000, C 0.000 }
gfCNCPoint5[15162] = {X 266.2556, Y 90.2554, Z -7.1667, A 0.000, B 0.000, C 0.000 }
gfCNCPoint5[15163] = {X 263.5102, Y 89.1792, Z -7.1667, A 0.000, B 0.000, C 0.000 }
gfCNCPoint5[15164] = {X 261.4785, Y 90.4951, Z -7.1667, A 0.000, B 0.000, C 0.000 }
gfCNCPoint5[15165] = {X 261.4785, Y 92.8951, Z -7.1667, A 0.000, B 0.000, C 0.000 }
gfCNCPoint5[15166] = {X 267.4973, Y 92.8951, Z -7.1667, A 0.000, B 0.000, C 0.000 }
gfCNCPoint5[15167] = {X 267.8429, Y 92.2376, Z -7.1667, A 0.000, B 0.000, C 0.000 }
gfCNCPoint5[15168] = {X 268.2378, Y 91.6085, Z -7.1667, A 0.000, B 0.000, C 0.000 }
gfCNCPoint5[15169] = {X 269.1700, Y 90.4463, Z -7.1667, A 0.000, B 0.000, C 0.000 }
gfCNCPoint5[15170] = {X 270.2694, Y 89.4409, Z -7.1667, A 0.000, B 0.000, C 0.000 }
gfCNCPoint5[15171] = {X 270.2694, Y 89.2510, Z -7.1667, A 0.000, B 0.000, C 0.000 }
gfCNCPoint5[15172] = {X 263.2393, Y 86.4951, Z -7.1667, A 0.000, B 0.000, C 0.000 }
gfCNCPoint5[15173] = {X 253.3586, Y 92.8951, Z -7.1667, A 0.000, B 0.000, C 0.000 }
gfCNCPoint5[15174] = {X 261.4785, Y 92.8951, Z -7.1667, A 0.000, B 0.000, C 0.000 }
gfCNCPoint5[15175] = {X 261.4785, Y 95.2951, Z -7.1667, A 0.000, B 0.000, C 0.000 }
gfCNCPoint5[15176] = {X 269.1713, Y 95.2951, Z -7.1667, A 0.000, B 0.000, C 0.000 }
gfCNCPoint5[15177] = {X 269.5515, Y 94.1745, Z -7.1667, A 0.000, B 0.000, C 0.000 }
gfCNCPoint5[15178] = {X 270.1082, Y 93.1304, Z -7.1667, A 0.000, B 0.000, C 0.000 }
gfCNCPoint5[15179] = {X 270.8267, Y 92.1901, Z -7.1667, A 0.000, B 0.000, C 0.000 }
gfCNCPoint5[15180] = {X 271.6880, Y 91.3787, Z -7.1667, A 0.000, B 0.000, C 0.000 }
gfCNCPoint5[15181] = {X 272.6694, Y 90.7176, Z -7.1667, A 0.000, B 0.000, C 0.000 }
gfCNCPoint5[15182] = {X 272.6694, Y 87.6139, Z -7.1667, A 0.000, B 0.000, C 0.000 }
gfCNCPoint5[15183] = {X 262.9684, Y 83.8111, Z -7.1667, A 0.000, B 0.000, C 0.000 }
gfCNCPoint5[15184] = {X 245.2387, Y 95.2951, Z -7.1667, A 0.000, B 0.000, C 0.000 }
gfCNCPoint5[15185] = {X 261.4785, Y 95.2951, Z -7.1667, A 0.000, B 0.000, C 0.000 }
gfCNCPoint5[15186] = {X 261.4785, Y 97.6951, Z -7.1667, A 0.000, B 0.000, C 0.000 }
gfCNCPoint5[15187] = {X 271.3527, Y 97.6951, Z -7.1667, A 0.000, B 0.000, C 0.000 }
gfCNCPoint5[15188] = {X 271.3529, Y 97.0186, Z -7.1667, A 0.000, B 0.000, C 0.000 }
gfCNCPoint5[15189] = {X 271.4810, Y 95.9545, Z -7.1667, A 0.000, B 0.000, C 0.000 }
gfCNCPoint5[15190] = {X 271.8382, Y 94.9440, Z -7.1667, A 0.000, B 0.000, C 0.000 }
gfCNCPoint5[15191] = {X 272.4074, Y 94.0359, Z -7.1667, A 0.000, B 0.000, C 0.000 }
gfCNCPoint5[15192] = {X 273.1610, Y 93.2739, Z -7.1667, A 0.000, B 0.000, C 0.000 }
gfCNCPoint5[15193] = {X 274.0629, Y 92.6949, Z -7.1667, A 0.000, B 0.000, C 0.000 }
gfCNCPoint5[15194] = {X 275.0694, Y 92.3266, Z -7.1667, A 0.000, B 0.000, C 0.000 }
gfCNCPoint5[15195] = {X 275.0694, Y 85.9769, Z -7.1667, A 0.000, B 0.000, C 0.000 }
gfCNCPoint5[15196] = {X 262.6993, Y 81.1279, Z -7.1667, A 0.000, B 0.000, C 0.000 }
gfCNCPoint5[15197] = {X 262.5799, Y 81.2033, Z -7.1667, A 0.000, B 0.000, C 0.000 }
gfCNCPoint5[15198] = {X 238.3589, Y 96.8918, Z -7.1667, A 0.000, B 0.000, C 0.000 }
gfCNCPoint5[15199] = {X 238.3598, Y 97.0659, Z -7.1667, A 0.000, B 0.000, C 0.000 }
gfCNCPoint5[15200] = {X 238.3598, Y 97.6951, Z -7.1667, A 0.000, B 0.000, C 0.000 }
gfCNCPoint5[15201] = {X 261.4785, Y 97.6951, Z -7.1667, A 0.000, B 0.000, C 0.000 }
gfCNCPoint5[15202] = {X 261.4785, Y 100.0951, Z -7.1667, A 0.000, B 0.000, C 0.000 }
gfCNCPoint5[15203] = {X 271.8253, Y 100.0951, Z -7.1667, A 0.000, B 0.000, C 0.000 }
gfCNCPoint5[15204] = {X 272.2941, Y 100.8813, Z -7.1667, A 0.000, B 0.000, C 0.000 }
gfCNCPoint5[15205] = {X 272.9014, Y 101.5661, Z -7.1667, A 0.000, B 0.000, C 0.000 }
gfCNCPoint5[15206] = {X 273.6260, Y 102.1254, Z -7.1667, A 0.000, B 0.000, C 0.000 }
gfCNCPoint5[15207] = {X 274.4422, Y 102.5397, Z -7.1667, A 0.000, B 0.000, C 0.000 }
gfCNCPoint5[15208] = {X 275.3214, Y 102.7942, Z -7.1667, A 0.000, B 0.000, C 0.000 }
gfCNCPoint5[15209] = {X 276.2327, Y 102.8800, Z -7.1667, A 0.000, B 0.000, C 0.000 }
gfCNCPoint5[15210] = {X 292.7731, Y 102.8800, Z -7.1667, A 0.000, B 0.000, C 0.000 }
gfCNCPoint5[15211] = {X 293.6844, Y 102.7942, Z -7.1667, A 0.000, B 0.000, C 0.000 }
gfCNCPoint5[15212] = {X 294.5636, Y 102.5397, Z -7.1667, A 0.000, B 0.000, C 0.000 }
gfCNCPoint5[15213] = {X 295.3798, Y 102.1254, Z -7.1667, A 0.000, B 0.000, C 0.000 }
gfCNCPoint5[15214] = {X 296.1043, Y 101.5661, Z -7.1667, A 0.000, B 0.000, C 0.000 }
gfCNCPoint5[15215] = {X 296.7117, Y 100.8813, Z -7.1667, A 0.000, B 0.000, C 0.000 }
gfCNCPoint5[15216] = {X 297.1804, Y 100.0951, Z -7.1667, A 0.000, B 0.000, C 0.000 }
gfCNCPoint5[15217] = {X 319.1322, Y 100.0951, Z -7.1667, A 0.000, B 0.000, C 0.000 }
gfCNCPoint5[15218] = {X 321.4359, Y 100.8683, Z -7.1667, A 0.000, B 0.000, C 0.000 }
gfCNCPoint5[15219] = {X 323.7822, Y 101.5005, Z -7.1667, A 0.000, B 0.000, C 0.000 }
gfCNCPoint5[15220] = {X 326.1625, Y 101.9896, Z -7.1667, A 0.000, B 0.000, C 0.000 }
gfCNCPoint5[15221] = {X 330.1024, Y 102.5991, Z -7.1667, A 0.000, B 0.000, C 0.000 }
gfCNCPoint5[15222] = {X 334.0643, Y 103.0435, Z -7.1667, A 0.000, B 0.000, C 0.000 }
gfCNCPoint5[15223] = {X 338.0414, Y 103.3221, Z -7.1667, A 0.000, B 0.000, C 0.000 }
gfCNCPoint5[15224] = {X 343.7799, Y 103.5427, Z -7.1667, A 0.000, B 0.000, C 0.000 }
gfCNCPoint5[15225] = {X 349.5224, Y 103.5878, Z -7.1667, A 0.000, B 0.000, C 0.000 }
gfCNCPoint5[15226] = {X 355.2637, Y 103.4573, Z -7.1667, A 0.000, B 0.000, C 0.000 }
gfCNCPoint5[15227] = {X 360.9983, Y 103.1515, Z -7.1667, A 0.000, B 0.000, C 0.000 }
gfCNCPoint5[15228] = {X 364.9924, Y 102.7829, Z -7.1667, A 0.000, B 0.000, C 0.000 }
gfCNCPoint5[15229] = {X 368.9635, Y 102.2185, Z -7.1667, A 0.000, B 0.000, C 0.000 }
gfCNCPoint5[15230] = {X 372.9022, Y 101.4598, Z -7.1667, A 0.000, B 0.000, C 0.000 }
gfCNCPoint5[15231] = {X 375.2301, Y 100.8566, Z -7.1667, A 0.000, B 0.000, C 0.000 }
gfCNCPoint5[15232] = {X 377.5111, Y 100.0951, Z -7.1667, A 0.000, B 0.000, C 0.000 }
gfCNCPoint5[15233] = {X 391.9986, Y 100.0951, Z -7.1667, A 0.000, B 0.000, C 0.000 }
gfCNCPoint5[15234] = {X 392.4674, Y 100.8813, Z -7.1667, A 0.000, B 0.000, C 0.000 }
gfCNCPoint5[15235] = {X 393.0747, Y 101.5661, Z -7.1667, A 0.000, B 0.000, C 0.000 }
gfCNCPoint5[15236] = {X 393.7992, Y 102.1254, Z -7.1667, A 0.000, B 0.000, C 0.000 }
gfCNCPoint5[15237] = {X 394.6154, Y 102.5397, Z -7.1667, A 0.000, B 0.000, C 0.000 }
gfCNCPoint5[15238] = {X 395.4947, Y 102.7942, Z -7.1667, A 0.000, B 0.000, C 0.000 }
gfCNCPoint5[15239] = {X 396.4059, Y 102.8800, Z -7.1667, A 0.000, B 0.000, C 0.000 }
gfCNCPoint5[15240] = {X 415.7067, Y 102.8800, Z -7.1667, A 0.000, B 0.000, C 0.000 }
gfCNCPoint5[15241] = {X 416.6180, Y 102.7942, Z -7.1667, A 0.000, B 0.000, C 0.000 }
gfCNCPoint5[15242] = {X 417.4972, Y 102.5397, Z -7.1667, A 0.000, B 0.000, C 0.000 }
gfCNCPoint5[15243] = {X 418.3134, Y 102.1254, Z -7.1667, A 0.000, B 0.000, C 0.000 }
gfCNCPoint5[15244] = {X 419.0380, Y 101.5661, Z -7.1667, A 0.000, B 0.000, C 0.000 }
gfCNCPoint5[15245] = {X 419.6453, Y 100.8813, Z -7.1667, A 0.000, B 0.000, C 0.000 }
gfCNCPoint5[15246] = {X 420.1141, Y 100.0951, Z -7.1667, A 0.000, B 0.000, C 0.000 }
gfCNCPoint5[15247] = {X 443.7041, Y 100.0951, Z -7.1667, A 0.000, B 0.000, C 0.000 }
gfCNCPoint5[15248] = {X 443.7041, Y 90.4951, Z -7.1667, A 0.000, B 0.000, C 0.000 }
gfCNCPoint5[15249] = {X 448.3230, Y 90.4951, Z -7.1667, A 0.000, B 0.000, C 0.000 }
gfCNCPoint5[15250] = {X 448.4020, Y 90.3748, Z -7.1667, A 0.000, B 0.000, C 0.000 }
gfCNCPoint5[15251] = {X 448.4825, Y 90.2554, Z -7.1667, A 0.000, B 0.000, C 0.000 }
gfCNCPoint5[15252] = {X 445.7362, Y 89.1788, Z -7.1667, A 0.000, B 0.000, C 0.000 }
gfCNCPoint5[15253] = {X 443.7041, Y 90.4951, Z -7.1667, A 0.000, B 0.000, C 0.000 }
gfCNCPoint5[15254] = {X 443.7041, Y 92.8951, Z -7.1667, A 0.000, B 0.000, C 0.000 }
gfCNCPoint5[15255] = {X 449.7242, Y 92.8951, Z -7.1667, A 0.000, B 0.000, C 0.000 }
gfCNCPoint5[15256] = {X 450.0698, Y 92.2376, Z -7.1667, A 0.000, B 0.000, C 0.000 }
gfCNCPoint5[15257] = {X 450.4647, Y 91.6084, Z -7.1667, A 0.000, B 0.000, C 0.000 }
gfCNCPoint5[15258] = {X 451.3969, Y 90.4463, Z -7.1667, A 0.000, B 0.000, C 0.000 }
gfCNCPoint5[15259] = {X 452.4963, Y 89.4409, Z -7.1667, A 0.000, B 0.000, C 0.000 }
gfCNCPoint5[15260] = {X 452.4963, Y 89.2510, Z -7.1667, A 0.000, B 0.000, C 0.000 }
gfCNCPoint5[15261] = {X 445.4653, Y 86.4948, Z -7.1667, A 0.000, B 0.000, C 0.000 }
gfCNCPoint5[15262] = {X 435.5847, Y 92.8951, Z -7.1667, A 0.000, B 0.000, C 0.000 }
gfCNCPoint5[15263] = {X 443.7041, Y 92.8951, Z -7.1667, A 0.000, B 0.000, C 0.000 }
gfCNCPoint5[15264] = {X 443.7041, Y 95.2951, Z -7.1667, A 0.000, B 0.000, C 0.000 }
gfCNCPoint5[15265] = {X 451.3983, Y 95.2951, Z -7.1667, A 0.000, B 0.000, C 0.000 }
gfCNCPoint5[15266] = {X 451.7784, Y 94.1745, Z -7.1667, A 0.000, B 0.000, C 0.000 }
gfCNCPoint5[15267] = {X 452.3351, Y 93.1304, Z -7.1667, A 0.000, B 0.000, C 0.000 }
gfCNCPoint5[15268] = {X 453.0536, Y 92.1901, Z -7.1667, A 0.000, B 0.000, C 0.000 }
gfCNCPoint5[15269] = {X 453.9149, Y 91.3787, Z -7.1667, A 0.000, B 0.000, C 0.000 }
gfCNCPoint5[15270] = {X 454.8963, Y 90.7176, Z -7.1667, A 0.000, B 0.000, C 0.000 }
gfCNCPoint5[15271] = {X 454.8963, Y 87.6139, Z -7.1667, A 0.000, B 0.000, C 0.000 }
gfCNCPoint5[15272] = {X 445.1943, Y 83.8108, Z -7.1667, A 0.000, B 0.000, C 0.000 }
gfCNCPoint5[15273] = {X 427.4652, Y 95.2951, Z -7.1667, A 0.000, B 0.000, C 0.000 }
gfCNCPoint5[15274] = {X 443.7041, Y 95.2951, Z -7.1667, A 0.000, B 0.000, C 0.000 }
gfCNCPoint5[15275] = {X 443.7041, Y 97.6951, Z -7.1667, A 0.000, B 0.000, C 0.000 }
gfCNCPoint5[15276] = {X 453.5796, Y 97.6951, Z -7.1667, A 0.000, B 0.000, C 0.000 }
gfCNCPoint5[15277] = {X 453.5796, Y 97.0659, Z -7.1667, A 0.000, B 0.000, C 0.000 }
gfCNCPoint5[15278] = {X 453.6990, Y 95.9930, Z -7.1667, A 0.000, B 0.000, C 0.000 }
gfCNCPoint5[15279] = {X 454.0514, Y 94.9725, Z -7.1667, A 0.000, B 0.000, C 0.000 }
gfCNCPoint5[15280] = {X 454.6196, Y 94.0545, Z -7.1667, A 0.000, B 0.000, C 0.000 }
gfCNCPoint5[15281] = {X 455.3757, Y 93.2839, Z -7.1667, A 0.000, B 0.000, C 0.000 }
gfCNCPoint5[15282] = {X 456.2827, Y 92.6984, Z -7.1667, A 0.000, B 0.000, C 0.000 }
gfCNCPoint5[15283] = {X 457.2963, Y 92.3266, Z -7.1667, A 0.000, B 0.000, C 0.000 }
gfCNCPoint5[15284] = {X 457.2963, Y 85.9769, Z -7.1667, A 0.000, B 0.000, C 0.000 }
gfCNCPoint5[15285] = {X 444.9234, Y 81.1267, Z -7.1667, A 0.000, B 0.000, C 0.000 }
gfCNCPoint5[15286] = {X 420.5858, Y 96.8919, Z -7.1667, A 0.000, B 0.000, C 0.000 }
gfCNCPoint5[15287] = {X 420.5867, Y 97.0659, Z -7.1667, A 0.000, B 0.000, C 0.000 }
gfCNCPoint5[15288] = {X 420.5867, Y 97.6951, Z -7.1667, A 0.000, B 0.000, C 0.000 }
gfCNCPoint5[15289] = {X 443.7041, Y 97.6951, Z -7.1667, A 0.000, B 0.000, C 0.000 }
gfCNCPoint5[15290] = {X 443.7041, Y 100.0951, Z -7.1667, A 0.000, B 0.000, C 0.000 }
gfCNCPoint5[15291] = {X 454.0522, Y 100.0951, Z -7.1667, A 0.000, B 0.000, C 0.000 }
gfCNCPoint5[15292] = {X 454.5210, Y 100.8813, Z -7.1667, A 0.000, B 0.000, C 0.000 }
gfCNCPoint5[15293] = {X 455.1283, Y 101.5661, Z -7.1667, A 0.000, B 0.000, C 0.000 }
gfCNCPoint5[15294] = {X 455.8529, Y 102.1254, Z -7.1667, A 0.000, B 0.000, C 0.000 }
gfCNCPoint5[15295] = {X 456.6691, Y 102.5397, Z -7.1667, A 0.000, B 0.000, C 0.000 }
gfCNCPoint5[15296] = {X 457.5483, Y 102.7942, Z -7.1667, A 0.000, B 0.000, C 0.000 }
gfCNCPoint5[15297] = {X 458.4596, Y 102.8800, Z -7.1667, A 0.000, B 0.000, C 0.000 }
gfCNCPoint5[15298] = {X 475.0000, Y 102.8800, Z -7.1667, A 0.000, B 0.000, C 0.000 }
gfCNCPoint5[15299] = {X 475.9113, Y 102.7942, Z -7.1667, A 0.000, B 0.000, C 0.000 }
gfCNCPoint5[15300] = {X 476.7905, Y 102.5397, Z -7.1667, A 0.000, B 0.000, C 0.000 }
gfCNCPoint5[15301] = {X 477.6067, Y 102.1254, Z -7.1667, A 0.000, B 0.000, C 0.000 }
gfCNCPoint5[15302] = {X 478.3313, Y 101.5661, Z -7.1667, A 0.000, B 0.000, C 0.000 }
gfCNCPoint5[15303] = {X 478.9386, Y 100.8813, Z -7.1667, A 0.000, B 0.000, C 0.000 }
gfCNCPoint5[15304] = {X 479.4074, Y 100.0951, Z -7.1667, A 0.000, B 0.000, C 0.000 }
gfCNCPoint5[15305] = {X 507.6812, Y 100.0951, Z -7.1667, A 0.000, B 0.000, C 0.000 }
gfCNCPoint5[15306] = {X 507.6812, Y 107.6951, Z -7.1667, A 0.000, B 0.000, C 0.000 }
gfCNCPoint5[15307] = {X 507.6812, Y 107.6951, Z -4.1667, A 0.000, B 0.000, C 0.000 }
gfCNCPoint5[15308] = {X 507.6812, Y 107.6951, Z 11.0000, A 0.000, B 0.000, C 0.000 }
gfCNCPoint5[15309] = {X 108.5570, Y 40.8974, Z 11.0000, A 0.000, B 0.000, C 0.000 }
gfCNCPoint5[15310] = {X 108.5570, Y 40.8974, Z -3.3333, A 0.000, B 0.000, C 0.000 }
gfCNCPoint5[15311] = {X 108.5570, Y 40.8974, Z -7.1667, A 0.000, B 0.000, C 0.000 }
gfCNCPoint5[15312] = {X 108.0692, Y 42.0895, Z -7.1667, A 0.000, B 0.000, C 0.000 }
gfCNCPoint5[15313] = {X 108.0970, Y 42.0413, Z -7.1667, A 0.000, B 0.000, C 0.000 }
gfCNCPoint5[15314] = {X 108.1254, Y 41.9933, Z -7.1667, A 0.000, B 0.000, C 0.000 }
gfCNCPoint5[15315] = {X 108.5484, Y 41.3819, Z -7.1667, A 0.000, B 0.000, C 0.000 }
gfCNCPoint5[15316] = {X 109.0449, Y 40.8286, Z -7.1667, A 0.000, B 0.000, C 0.000 }
gfCNCPoint5[15317] = {X 109.0448, Y 39.7052, Z -7.1667, A 0.000, B 0.000, C 0.000 }
gfCNCPoint5[15318] = {X 108.5570, Y 40.8974, Z -7.1667, A 0.000, B 0.000, C 0.000 }
gfCNCPoint5[15319] = {X 108.5570, Y 40.8974, Z -4.1667, A 0.000, B 0.000, C 0.000 }
gfCNCPoint5[15320] = {X 108.5570, Y 40.8974, Z 11.0000, A 0.000, B 0.000, C 0.000 }
gfCNCPoint5[15321] = {X 95.6823, Y 40.8712, Z 11.0000, A 0.000, B 0.000, C 0.000 }
gfCNCPoint5[15322] = {X 95.6823, Y 40.8712, Z -3.3333, A 0.000, B 0.000, C 0.000 }
gfCNCPoint5[15323] = {X 95.6823, Y 40.8712, Z -7.1667, A 0.000, B 0.000, C 0.000 }
gfCNCPoint5[15324] = {X 95.2120, Y 39.7212, Z -7.1667, A 0.000, B 0.000, C 0.000 }
gfCNCPoint5[15325] = {X 95.2120, Y 40.8682, Z -7.1667, A 0.000, B 0.000, C 0.000 }
gfCNCPoint5[15326] = {X 95.7305, Y 41.4054, Z -7.1667, A 0.000, B 0.000, C 0.000 }
gfCNCPoint5[15327] = {X 96.1525, Y 42.0213, Z -7.1667, A 0.000, B 0.000, C 0.000 }
gfCNCPoint5[15328] = {X 95.6823, Y 40.8712, Z -7.1667, A 0.000, B 0.000, C 0.000 }
gfCNCPoint5[15329] = {X 95.6823, Y 40.8712, Z -4.1667, A 0.000, B 0.000, C 0.000 }
gfCNCPoint5[15330] = {X 95.6823, Y 40.8712, Z 11.0000, A 0.000, B 0.000, C 0.000 }
gfCNCPoint5[15331] = {X -7.6967, Y 43.2749, Z 11.0000, A 0.000, B 0.000, C 0.000 }
gfCNCPoint5[15332] = {X -7.6967, Y 43.2749, Z -4.1667, A 0.000, B 0.000, C 0.000 }
gfCNCPoint5[15333] = {X -7.6967, Y 43.2749, Z -7.1667, A 0.000, B 0.000, C 0.000 }
gfCNCPoint5[15334] = {X -3.6967, Y 30.7981, Z -7.1667, A 0.000, B 0.000, C 0.000 }
gfCNCPoint5[15335] = {X -3.5211, Y 30.2831, Z -7.1667, A 0.000, B 0.000, C 0.000 }
gfCNCPoint5[15336] = {X -3.3269, Y 29.7749, Z -7.1667, A 0.000, B 0.000, C 0.000 }
gfCNCPoint5[15337] = {X -2.7038, Y 28.4548, Z -7.1667, A 0.000, B 0.000, C 0.000 }
gfCNCPoint5[15338] = {X -1.9100, Y 27.2298, Z -7.1667, A 0.000, B 0.000, C 0.000 }
gfCNCPoint5[15339] = {X -0.9598, Y 26.1217, Z -7.1667, A 0.000, B 0.000, C 0.000 }
gfCNCPoint5[15340] = {X 0.1299, Y 25.1504, Z -7.1667, A 0.000, B 0.000, C 0.000 }
gfCNCPoint5[15341] = {X 1.3395, Y 24.3332, Z -7.1667, A 0.000, B 0.000, C 0.000 }
gfCNCPoint5[15342] = {X 0.5792, Y 23.9229, Z -7.1667, A 0.000, B 0.000, C 0.000 }
gfCNCPoint5[15343] = {X -0.0861, Y 23.3720, Z -7.1667, A 0.000, B 0.000, C 0.000 }
gfCNCPoint5[15344] = {X -0.6311, Y 22.7017, Z -7.1667, A 0.000, B 0.000, C 0.000 }
gfCNCPoint5[15345] = {X -1.0345, Y 21.9379, Z -7.1667, A 0.000, B 0.000, C 0.000 }
gfCNCPoint5[15346] = {X -3.6458, Y 15.5423, Z -7.1667, A 0.000, B 0.000, C 0.000 }
gfCNCPoint5[15347] = {X -3.6717, Y 15.4772, Z -7.1667, A 0.000, B 0.000, C 0.000 }
gfCNCPoint5[15348] = {X -3.6967, Y 15.4117, Z -7.1667, A 0.000, B 0.000, C 0.000 }
gfCNCPoint5[15349] = {X -7.6967, Y 4.6474, Z -7.1667, A 0.000, B 0.000, C 0.000 }
gfCNCPoint5[15350] = {X -7.6967, Y 4.6474, Z -4.1667, A 0.000, B 0.000, C 0.000 }
gfCNCPoint5[15351] = {X -7.6967, Y 4.6474, Z 11.0000, A 0.000, B 0.000, C 0.000 }
gfCNCPoint5[15352] = {X -7.6967, Y 16.4130, Z 11.0000, A 0.000, B 0.000, C 0.000 }
gfCNCPoint5[15353] = {X -7.6967, Y 16.4130, Z -4.1667, A 0.000, B 0.000, C 0.000 }
gfCNCPoint5[15354] = {X -7.6967, Y 16.4130, Z -7.1667, A 0.000, B 0.000, C 0.000 }
gfCNCPoint5[15355] = {X -4.8865, Y 16.4130, Z -7.1667, A 0.000, B 0.000, C 0.000 }
gfCNCPoint5[15356] = {X -3.6967, Y 12.5941, Z -7.1667, A 0.000, B 0.000, C 0.000 }
gfCNCPoint5[15357] = {X -3.6606, Y 12.4837, Z -7.1667, A 0.000, B 0.000, C 0.000 }
gfCNCPoint5[15358] = {X -3.6217, Y 12.3744, Z -7.1667, A 0.000, B 0.000, C 0.000 }
gfCNCPoint5[15359] = {X -3.1668, Y 11.4829, Z -7.1667, A 0.000, B 0.000, C 0.000 }
gfCNCPoint5[15360] = {X -2.5189, Y 10.7201, Z -7.1667, A 0.000, B 0.000, C 0.000 }
gfCNCPoint5[15361] = {X -1.7129, Y 10.1268, Z -7.1667, A 0.000, B 0.000, C 0.000 }
gfCNCPoint5[15362] = {X -1.1156, Y 9.7861, Z -7.1667, A 0.000, B 0.000, C 0.000 }
gfCNCPoint5[15363] = {X -0.2328, Y 9.4056, Z -7.1667, A 0.000, B 0.000, C 0.000 }
gfCNCPoint5[15364] = {X 0.7123, Y 9.2298, Z -7.1667, A 0.000, B 0.000, C 0.000 }
gfCNCPoint5[15365] = {X 1.6728, Y 9.2673, Z -7.1667, A 0.000, B 0.000, C 0.000 }
gfCNCPoint5[15366] = {X 2.6013, Y 9.5164, Z -7.1667, A 0.000, B 0.000, C 0.000 }
gfCNCPoint5[15367] = {X 3.4887, Y 9.1194, Z -7.1667, A 0.000, B 0.000, C 0.000 }
gfCNCPoint5[15368] = {X 5.5657, Y 8.3368, Z -7.1667, A 0.000, B 0.000, C 0.000 }
gfCNCPoint5[15369] = {X 7.7065, Y 7.7511, Z -7.1667, A 0.000, B 0.000, C 0.000 }
gfCNCPoint5[15370] = {X 9.8926, Y 7.3673, Z -7.1667, A 0.000, B 0.000, C 0.000 }
gfCNCPoint5[15371] = {X 12.1050, Y 7.1889, Z -7.1667, A 0.000, B 0.000, C 0.000 }
gfCNCPoint5[15372] = {X 14.3243, Y 7.2173, Z -7.1667, A 0.000, B 0.000, C 0.000 }
gfCNCPoint5[15373] = {X 16.5314, Y 7.4523, Z -7.1667, A 0.000, B 0.000, C 0.000 }
gfCNCPoint5[15374] = {X 18.2667, Y 7.8077, Z -7.1667, A 0.000, B 0.000, C 0.000 }
gfCNCPoint5[15375] = {X 19.9571, Y 8.3372, Z -7.1667, A 0.000, B 0.000, C 0.000 }
gfCNCPoint5[15376] = {X 21.5850, Y 9.0354, Z -7.1667, A 0.000, B 0.000, C 0.000 }
gfCNCPoint5[15377] = {X 23.1338, Y 9.8951, Z -7.1667, A 0.000, B 0.000, C 0.000 }
gfCNCPoint5[15378] = {X 24.5873, Y 10.9073, Z -7.1667, A 0.000, B 0.000, C 0.000 }
gfCNCPoint5[15379] = {X 25.6728, Y 11.8564, Z -7.1667, A 0.000, B 0.000, C 0.000 }
gfCNCPoint5[15380] = {X 26.6465, Y 12.9198, Z -7.1667, A 0.000, B 0.000, C 0.000 }
gfCNCPoint5[15381] = {X 27.4965, Y 14.0845, Z -7.1667, A 0.000, B 0.000, C 0.000 }
gfCNCPoint5[15382] = {X 28.2123, Y 15.3361, Z -7.1667, A 0.000, B 0.000, C 0.000 }
gfCNCPoint5[15383] = {X 28.7852, Y 16.6593, Z -7.1667, A 0.000, B 0.000, C 0.000 }
gfCNCPoint5[15384] = {X 29.2600, Y 18.3155, Z -7.1667, A 0.000, B 0.000, C 0.000 }
gfCNCPoint5[15385] = {X 29.5417, Y 20.0153, Z -7.1667, A 0.000, B 0.000, C 0.000 }
gfCNCPoint5[15386] = {X 29.6268, Y 21.7361, Z -7.1667, A 0.000, B 0.000, C 0.000 }
gfCNCPoint5[15387] = {X 29.5140, Y 23.4553, Z -7.1667, A 0.000, B 0.000, C 0.000 }
gfCNCPoint5[15388] = {X 29.2049, Y 25.1502, Z -7.1667, A 0.000, B 0.000, C 0.000 }
gfCNCPoint5[15389] = {X 28.7625, Y 26.5966, Z -7.1667, A 0.000, B 0.000, C 0.000 }
gfCNCPoint5[15390] = {X 28.1371, Y 27.9738, Z -7.1667, A 0.000, B 0.000, C 0.000 }
gfCNCPoint5[15391] = {X 27.3392, Y 29.2588, Z -7.1667, A 0.000, B 0.000, C 0.000 }
gfCNCPoint5[15392] = {X 26.3821, Y 30.4300, Z -7.1667, A 0.000, B 0.000, C 0.000 }
gfCNCPoint5[15393] = {X 25.2818, Y 31.4678, Z -7.1667, A 0.000, B 0.000, C 0.000 }
gfCNCPoint5[15394] = {X 26.0856, Y 31.8100, Z -7.1667, A 0.000, B 0.000, C 0.000 }
gfCNCPoint5[15395] = {X 26.8042, Y 32.3069, Z -7.1667, A 0.000, B 0.000, C 0.000 }
gfCNCPoint5[15396] = {X 27.4081, Y 32.9382, Z -7.1667, A 0.000, B 0.000, C 0.000 }
gfCNCPoint5[15397] = {X 27.8726, Y 33.6781, Z -7.1667, A 0.000, B 0.000, C 0.000 }
gfCNCPoint5[15398] = {X 30.9100, Y 39.9530, Z -7.1667, A 0.000, B 0.000, C 0.000 }
gfCNCPoint5[15399] = {X 31.2306, Y 40.8622, Z -7.1667, A 0.000, B 0.000, C 0.000 }
gfCNCPoint5[15400] = {X 31.3415, Y 41.8197, Z -7.1667, A 0.000, B 0.000, C 0.000 }
gfCNCPoint5[15401] = {X 31.2374, Y 42.7781, Z -7.1667, A 0.000, B 0.000, C 0.000 }
gfCNCPoint5[15402] = {X 30.9234, Y 43.6895, Z -7.1667, A 0.000, B 0.000, C 0.000 }
gfCNCPoint5[15403] = {X 30.4150, Y 44.5085, Z -7.1667, A 0.000, B 0.000, C 0.000 }
gfCNCPoint5[15404] = {X 29.7377, Y 45.1945, Z -7.1667, A 0.000, B 0.000, C 0.000 }
gfCNCPoint5[15405] = {X 29.2017, Y 45.6278, Z -7.1667, A 0.000, B 0.000, C 0.000 }
gfCNCPoint5[15406] = {X 28.4980, Y 46.0916, Z -7.1667, A 0.000, B 0.000, C 0.000 }
gfCNCPoint5[15407] = {X 27.7177, Y 46.4103, Z -7.1667, A 0.000, B 0.000, C 0.000 }
gfCNCPoint5[15408] = {X 26.8904, Y 46.5718, Z -7.1667, A 0.000, B 0.000, C 0.000 }
gfCNCPoint5[15409] = {X 26.0476, Y 46.5700, Z -7.1667, A 0.000, B 0.000, C 0.000 }
gfCNCPoint5[15410] = {X 25.2210, Y 46.4049, Z -7.1667, A 0.000, B 0.000, C 0.000 }
gfCNCPoint5[15411] = {X 23.4205, Y 47.3551, Z -7.1667, A 0.000, B 0.000, C 0.000 }
gfCNCPoint5[15412] = {X 21.5582, Y 48.1776, Z -7.1667, A 0.000, B 0.000, C 0.000 }
gfCNCPoint5[15413] = {X 19.6432, Y 48.8684, Z -7.1667, A 0.000, B 0.000, C 0.000 }
gfCNCPoint5[15414] = {X 17.7035, Y 49.4158, Z -7.1667, A 0.000, B 0.000, C 0.000 }
gfCNCPoint5[15415] = {X 15.7230, Y 49.7895, Z -7.1667, A 0.000, B 0.000, C 0.000 }
gfCNCPoint5[15416] = {X 13.7171, Y 49.9865, Z -7.1667, A 0.000, B 0.000, C 0.000 }
gfCNCPoint5[15417] = {X 11.7017, Y 50.0052, Z -7.1667, A 0.000, B 0.000, C 0.000 }
gfCNCPoint5[15418] = {X 9.6926, Y 49.8456, Z -7.1667, A 0.000, B 0.000, C 0.000 }
gfCNCPoint5[15419] = {X 7.7054, Y 49.5088, Z -7.1667, A 0.000, B 0.000, C 0.000 }
gfCNCPoint5[15420] = {X 5.8040, Y 48.9878, Z -7.1667, A 0.000, B 0.000, C 0.000 }
gfCNCPoint5[15421] = {X 3.9771, Y 48.2467, Z -7.1667, A 0.000, B 0.000, C 0.000 }
gfCNCPoint5[15422] = {X 2.2501, Y 47.2956, Z -7.1667, A 0.000, B 0.000, C 0.000 }
gfCNCPoint5[15423] = {X 0.6472, Y 46.1478, Z -7.1667, A 0.000, B 0.000, C 0.000 }
gfCNCPoint5[15424] = {X -0.4850, Y 45.1299, Z -7.1667, A 0.000, B 0.000, C 0.000 }
gfCNCPoint5[15425] = {X -1.4907, Y 43.9867, Z -7.1667, A 0.000, B 0.000, C 0.000 }
gfCNCPoint5[15426] = {X -2.3560, Y 42.7340, Z -7.1667, A 0.000, B 0.000, C 0.000 }
gfCNCPoint5[15427] = {X -3.0692, Y 41.3889, Z -7.1667, A 0.000, B 0.000, C 0.000 }
gfCNCPoint5[15428] = {X -3.6205, Y 39.9697, Z -7.1667, A 0.000, B 0.000, C 0.000 }
gfCNCPoint5[15429] = {X -3.6592, Y 39.8478, Z -7.1667, A 0.000, B 0.000, C 0.000 }
gfCNCPoint5[15430] = {X -3.6967, Y 39.7255, Z -7.1667, A 0.000, B 0.000, C 0.000 }
gfCNCPoint5[15431] = {X -4.8496, Y 35.8952, Z -7.1667, A 0.000, B 0.000, C 0.000 }
gfCNCPoint5[15432] = {X -7.9952, Y 36.0087, Z -7.1667, A 0.000, B 0.000, C 0.000 }
gfCNCPoint5[15433] = {X -7.9952, Y 36.0087, Z -4.1667, A 0.000, B 0.000, C 0.000 }
gfCNCPoint5[15434] = {X -7.9952, Y 36.0087, Z 11.0000, A 0.000, B 0.000, C 0.000 }
gfCNCPoint5[15435] = {X 608.0000, Y 40.1190, Z 11.0000, A 0.000, B 0.000, C 0.000 }
gfCNCPoint5[15436] = {X 608.0000, Y 40.1190, Z -4.1667, A 0.000, B 0.000, C 0.000 }
gfCNCPoint5[15437] = {X 608.0000, Y 40.1190, Z -7.1667, A 0.000, B 0.000, C 0.000 }
gfCNCPoint5[15438] = {X 603.6967, Y 47.2354, Z -7.1667, A 0.000, B 0.000, C 0.000 }
gfCNCPoint5[15439] = {X 603.6635, Y 47.2894, Z -7.1667, A 0.000, B 0.000, C 0.000 }
gfCNCPoint5[15440] = {X 603.6295, Y 47.3430, Z -7.1667, A 0.000, B 0.000, C 0.000 }
gfCNCPoint5[15441] = {X 603.0931, Y 48.0158, Z -7.1667, A 0.000, B 0.000, C 0.000 }
gfCNCPoint5[15442] = {X 602.4340, Y 48.5690, Z -7.1667, A 0.000, B 0.000, C 0.000 }
gfCNCPoint5[15443] = {X 601.6784, Y 48.9806, Z -7.1667, A 0.000, B 0.000, C 0.000 }
gfCNCPoint5[15444] = {X 600.8562, Y 49.2343, Z -7.1667, A 0.000, B 0.000, C 0.000 }
gfCNCPoint5[15445] = {X 600.0000, Y 49.3200, Z -7.1667, A 0.000, B 0.000, C 0.000 }
gfCNCPoint5[15446] = {X 593.5565, Y 49.3200, Z -7.1667, A 0.000, B 0.000, C 0.000 }
gfCNCPoint5[15447] = {X 592.5952, Y 49.2117, Z -7.1667, A 0.000, B 0.000, C 0.000 }
gfCNCPoint5[15448] = {X 591.6822, Y 48.8922, Z -7.1667, A 0.000, B 0.000, C 0.000 }
gfCNCPoint5[15449] = {X 590.8631, Y 48.3775, Z -7.1667, A 0.000, B 0.000, C 0.000 }
gfCNCPoint5[15450] = {X 590.1790, Y 47.6935, Z -7.1667, A 0.000, B 0.000, C 0.000 }
gfCNCPoint5[15451] = {X 589.6643, Y 46.8744, Z -7.1667, A 0.000, B 0.000, C 0.000 }
gfCNCPoint5[15452] = {X 589.3448, Y 45.9613, Z -7.1667, A 0.000, B 0.000, C 0.000 }
gfCNCPoint5[15453] = {X 589.2365, Y 45.0000, Z -7.1667, A 0.000, B 0.000, C 0.000 }
gfCNCPoint5[15454] = {X 589.2365, Y 44.0647, Z -7.1667, A 0.000, B 0.000, C 0.000 }
gfCNCPoint5[15455] = {X 589.3403, Y 43.1364, Z -7.1667, A 0.000, B 0.000, C 0.000 }
gfCNCPoint5[15456] = {X 589.6396, Y 42.2515, Z -7.1667, A 0.000, B 0.000, C 0.000 }
gfCNCPoint5[15457] = {X 590.1206, Y 41.4507, Z -7.1667, A 0.000, B 0.000, C 0.000 }
gfCNCPoint5[15458] = {X 590.7612, Y 40.7709, Z -7.1667, A 0.000, B 0.000, C 0.000 }
gfCNCPoint5[15459] = {X 590.7619, Y 33.5330, Z -7.1667, A 0.000, B 0.000, C 0.000 }
gfCNCPoint5[15460] = {X 585.4453, Y 46.6524, Z -7.1667, A 0.000, B 0.000, C 0.000 }
gfCNCPoint5[15461] = {X 585.0755, Y 47.3550, Z -7.1667, A 0.000, B 0.000, C 0.000 }
gfCNCPoint5[15462] = {X 584.5834, Y 47.9780, Z -7.1667, A 0.000, B 0.000, C 0.000 }
gfCNCPoint5[15463] = {X 583.9856, Y 48.5004, Z -7.1667, A 0.000, B 0.000, C 0.000 }
gfCNCPoint5[15464] = {X 583.3023, Y 48.9046, Z -7.1667, A 0.000, B 0.000, C 0.000 }
gfCNCPoint5[15465] = {X 582.3585, Y 49.2242, Z -7.1667, A 0.000, B 0.000, C 0.000 }
gfCNCPoint5[15466] = {X 581.3666, Y 49.3191, Z -7.1667, A 0.000, B 0.000, C 0.000 }
gfCNCPoint5[15467] = {X 580.3794, Y 49.1842, Z -7.1667, A 0.000, B 0.000, C 0.000 }
gfCNCPoint5[15468] = {X 579.4493, Y 48.8268, Z -7.1667, A 0.000, B 0.000, C 0.000 }
gfCNCPoint5[15469] = {X 578.6259, Y 48.2657, Z -7.1667, A 0.000, B 0.000, C 0.000 }
gfCNCPoint5[15470] = {X 577.9529, Y 47.5309, Z -7.1667, A 0.000, B 0.000, C 0.000 }
gfCNCPoint5[15471] = {X 577.4662, Y 46.6615, Z -7.1667, A 0.000, B 0.000, C 0.000 }
gfCNCPoint5[15472] = {X 572.0199, Y 33.3439, Z -7.1667, A 0.000, B 0.000, C 0.000 }
gfCNCPoint5[15473] = {X 572.0201, Y 40.7713, Z -7.1667, A 0.000, B 0.000, C 0.000 }
gfCNCPoint5[15474] = {X 572.6580, Y 41.4422, Z -7.1667, A 0.000, B 0.000, C 0.000 }
gfCNCPoint5[15475] = {X 573.1384, Y 42.2336, Z -7.1667, A 0.000, B 0.000, C 0.000 }
gfCNCPoint5[15476] = {X 573.4390, Y 43.1092, Z -7.1667, A 0.000, B 0.000, C 0.000 }
gfCNCPoint5[15477] = {X 573.5463, Y 44.0287, Z -7.1667, A 0.000, B 0.000, C 0.000 }
gfCNCPoint5[15478] = {X 573.5464, Y 45.0000, Z -7.1667, A 0.000, B 0.000, C 0.000 }
gfCNCPoint5[15479] = {X 573.4381, Y 45.9613, Z -7.1667, A 0.000, B 0.000, C 0.000 }
gfCNCPoint5[15480] = {X 573.1186, Y 46.8744, Z -7.1667, A 0.000, B 0.000, C 0.000 }
gfCNCPoint5[15481] = {X 572.6039, Y 47.6935, Z -7.1667, A 0.000, B 0.000, C 0.000 }
gfCNCPoint5[15482] = {X 571.9199, Y 48.3775, Z -7.1667, A 0.000, B 0.000, C 0.000 }
gfCNCPoint5[15483] = {X 571.1008, Y 48.8922, Z -7.1667, A 0.000, B 0.000, C 0.000 }
gfCNCPoint5[15484] = {X 570.1877, Y 49.2117, Z -7.1667, A 0.000, B 0.000, C 0.000 }
gfCNCPoint5[15485] = {X 569.2264, Y 49.3200, Z -7.1667, A 0.000, B 0.000, C 0.000 }
gfCNCPoint5[15486] = {X 562.4443, Y 49.3200, Z -7.1667, A 0.000, B 0.000, C 0.000 }
gfCNCPoint5[15487] = {X 561.4830, Y 49.2117, Z -7.1667, A 0.000, B 0.000, C 0.000 }
gfCNCPoint5[15488] = {X 560.5699, Y 48.8922, Z -7.1667, A 0.000, B 0.000, C 0.000 }
gfCNCPoint5[15489] = {X 559.7508, Y 48.3775, Z -7.1667, A 0.000, B 0.000, C 0.000 }
gfCNCPoint5[15490] = {X 559.0668, Y 47.6935, Z -7.1667, A 0.000, B 0.000, C 0.000 }
gfCNCPoint5[15491] = {X 558.5521, Y 46.8744, Z -7.1667, A 0.000, B 0.000, C 0.000 }
gfCNCPoint5[15492] = {X 558.2326, Y 45.9613, Z -7.1667, A 0.000, B 0.000, C 0.000 }
gfCNCPoint5[15493] = {X 558.1243, Y 45.0000, Z -7.1667, A 0.000, B 0.000, C 0.000 }
gfCNCPoint5[15494] = {X 558.1243, Y 44.0649, Z -7.1667, A 0.000, B 0.000, C 0.000 }
gfCNCPoint5[15495] = {X 558.2278, Y 43.1360, Z -7.1667, A 0.000, B 0.000, C 0.000 }
gfCNCPoint5[15496] = {X 558.5274, Y 42.2508, Z -7.1667, A 0.000, B 0.000, C 0.000 }
gfCNCPoint5[15497] = {X 559.0092, Y 41.4499, Z -7.1667, A 0.000, B 0.000, C 0.000 }
gfCNCPoint5[15498] = {X 559.6509, Y 40.7704, Z -7.1667, A 0.000, B 0.000, C 0.000 }
gfCNCPoint5[15499] = {X 559.6510, Y 9.2295, Z -7.1667, A 0.000, B 0.000, C 0.000 }
gfCNCPoint5[15500] = {X 559.0129, Y 8.5586, Z -7.1667, A 0.000, B 0.000, C 0.000 }
gfCNCPoint5[15501] = {X 558.5325, Y 7.7671, Z -7.1667, A 0.000, B 0.000, C 0.000 }
gfCNCPoint5[15502] = {X 558.2317, Y 6.8915, Z -7.1667, A 0.000, B 0.000, C 0.000 }
gfCNCPoint5[15503] = {X 558.1245, Y 5.9718, Z -7.1667, A 0.000, B 0.000, C 0.000 }
gfCNCPoint5[15504] = {X 558.1243, Y 5.0000, Z -7.1667, A 0.000, B 0.000, C 0.000 }
gfCNCPoint5[15505] = {X 558.2326, Y 4.0387, Z -7.1667, A 0.000, B 0.000, C 0.000 }
gfCNCPoint5[15506] = {X 558.5521, Y 3.1256, Z -7.1667, A 0.000, B 0.000, C 0.000 }
gfCNCPoint5[15507] = {X 559.0668, Y 2.3065, Z -7.1667, A 0.000, B 0.000, C 0.000 }
gfCNCPoint5[15508] = {X 559.7508, Y 1.6225, Z -7.1667, A 0.000, B 0.000, C 0.000 }
gfCNCPoint5[15509] = {X 560.5699, Y 1.1078, Z -7.1667, A 0.000, B 0.000, C 0.000 }
gfCNCPoint5[15510] = {X 561.4830, Y 0.7883, Z -7.1667, A 0.000, B 0.000, C 0.000 }
gfCNCPoint5[15511] = {X 562.4443, Y 0.6800, Z -7.1667, A 0.000, B 0.000, C 0.000 }
gfCNCPoint5[15512] = {X 570.9376, Y 0.6800, Z -7.1667, A 0.000, B 0.000, C 0.000 }
gfCNCPoint5[15513] = {X 571.8988, Y 0.7883, Z -7.1667, A 0.000, B 0.000, C 0.000 }
gfCNCPoint5[15514] = {X 572.8119, Y 1.1078, Z -7.1667, A 0.000, B 0.000, C 0.000 }
gfCNCPoint5[15515] = {X 573.6310, Y 1.6225, Z -7.1667, A 0.000, B 0.000, C 0.000 }
gfCNCPoint5[15516] = {X 574.3151, Y 2.3065, Z -7.1667, A 0.000, B 0.000, C 0.000 }
gfCNCPoint5[15517] = {X 574.8297, Y 3.1256, Z -7.1667, A 0.000, B 0.000, C 0.000 }
gfCNCPoint5[15518] = {X 575.1492, Y 4.0387, Z -7.1667, A 0.000, B 0.000, C 0.000 }
gfCNCPoint5[15519] = {X 575.2576, Y 5.0000, Z -7.1667, A 0.000, B 0.000, C 0.000 }
gfCNCPoint5[15520] = {X 575.2576, Y 5.9343, Z -7.1667, A 0.000, B 0.000, C 0.000 }
gfCNCPoint5[15521] = {X 575.1836, Y 6.7302, Z -7.1667, A 0.000, B 0.000, C 0.000 }
gfCNCPoint5[15522] = {X 574.9642, Y 7.4988, Z -7.1667, A 0.000, B 0.000, C 0.000 }
gfCNCPoint5[15523] = {X 574.6070, Y 8.2139, Z -7.1667, A 0.000, B 0.000, C 0.000 }
gfCNCPoint5[15524] = {X 581.1910, Y 24.3688, Z -7.1667, A 0.000, B 0.000, C 0.000 }
gfCNCPoint5[15525] = {X 587.8455, Y 8.0937, Z -7.1667, A 0.000, B 0.000, C 0.000 }
gfCNCPoint5[15526] = {X 587.5316, Y 7.4227, Z -7.1667, A 0.000, B 0.000, C 0.000 }
gfCNCPoint5[15527] = {X 587.3368, Y 6.7080, Z -7.1667, A 0.000, B 0.000, C 0.000 }
gfCNCPoint5[15528] = {X 587.2671, Y 5.9705, Z -7.1667, A 0.000, B 0.000, C 0.000 }
gfCNCPoint5[15529] = {X 587.2670, Y 5.0000, Z -7.1667, A 0.000, B 0.000, C 0.000 }
gfCNCPoint5[15530] = {X 587.3753, Y 4.0387, Z -7.1667, A 0.000, B 0.000, C 0.000 }
gfCNCPoint5[15531] = {X 587.6948, Y 3.1256, Z -7.1667, A 0.000, B 0.000, C 0.000 }
gfCNCPoint5[15532] = {X 588.2094, Y 2.3065, Z -7.1667, A 0.000, B 0.000, C 0.000 }
gfCNCPoint5[15533] = {X 588.8935, Y 1.6225, Z -7.1667, A 0.000, B 0.000, C 0.000 }
gfCNCPoint5[15534] = {X 589.7126, Y 1.1078, Z -7.1667, A 0.000, B 0.000, C 0.000 }
gfCNCPoint5[15535] = {X 590.6257, Y 0.7883, Z -7.1667, A 0.000, B 0.000, C 0.000 }
gfCNCPoint5[15536] = {X 591.5870, Y 0.6800, Z -7.1667, A 0.000, B 0.000, C 0.000 }
gfCNCPoint5[15537] = {X 600.0000, Y 0.6800, Z -7.1667, A 0.000, B 0.000, C 0.000 }
gfCNCPoint5[15538] = {X 600.8562, Y 0.7657, Z -7.1667, A 0.000, B 0.000, C 0.000 }
gfCNCPoint5[15539] = {X 601.6784, Y 1.0194, Z -7.1667, A 0.000, B 0.000, C 0.000 }
gfCNCPoint5[15540] = {X 602.4340, Y 1.4310, Z -7.1667, A 0.000, B 0.000, C 0.000 }
gfCNCPoint5[15541] = {X 603.0931, Y 1.9842, Z -7.1667, A 0.000, B 0.000, C 0.000 }
gfCNCPoint5[15542] = {X 603.6295, Y 2.6570, Z -7.1667, A 0.000, B 0.000, C 0.000 }
gfCNCPoint5[15543] = {X 603.6635, Y 2.7106, Z -7.1667, A 0.000, B 0.000, C 0.000 }
gfCNCPoint5[15544] = {X 603.6967, Y 2.7646, Z -7.1667, A 0.000, B 0.000, C 0.000 }
gfCNCPoint5[15545] = {X 608.0000, Y 9.8810, Z -7.1667, A 0.000, B 0.000, C 0.000 }
gfCNCPoint5[15546] = {X 608.0000, Y 9.8810, Z -4.1667, A 0.000, B 0.000, C 0.000 }
gfCNCPoint5[15547] = {X 608.0000, Y 9.8810, Z 11.0000, A 0.000, B 0.000, C 0.000 }
gfCNCPoint5[15548] = {X -7.6967, Y 16.7870, Z 11.0000, A 0.000, B 0.000, C 0.000 }
gfCNCPoint5[15549] = {X -7.6967, Y 16.7870, Z -4.1667, A 0.000, B 0.000, C 0.000 }
gfCNCPoint5[15550] = {X -7.6967, Y 16.7870, Z -7.1667, A 0.000, B 0.000, C 0.000 }
gfCNCPoint5[15551] = {X -4.6241, Y 16.7870, Z -7.1667, A 0.000, B 0.000, C 0.000 }
gfCNCPoint5[15552] = {X -3.6967, Y 12.8960, Z -7.1667, A 0.000, B 0.000, C 0.000 }
gfCNCPoint5[15553] = {X -3.6292, Y 12.6468, Z -7.1667, A 0.000, B 0.000, C 0.000 }
gfCNCPoint5[15554] = {X -3.5467, Y 12.4022, Z -7.1667, A 0.000, B 0.000, C 0.000 }
gfCNCPoint5[15555] = {X -3.1002, Y 11.5273, Z -7.1667, A 0.000, B 0.000, C 0.000 }
gfCNCPoint5[15556] = {X -2.4644, Y 10.7786, Z -7.1667, A 0.000, B 0.000, C 0.000 }
gfCNCPoint5[15557] = {X -1.6733, Y 10.1963, Z -7.1667, A 0.000, B 0.000, C 0.000 }
gfCNCPoint5[15558] = {X -1.0760, Y 9.8556, Z -7.1667, A 0.000, B 0.000, C 0.000 }
gfCNCPoint5[15559] = {X -0.2015, Y 9.4797, Z -7.1667, A 0.000, B 0.000, C 0.000 }
gfCNCPoint5[15560] = {X 0.7347, Y 9.3084, Z -7.1667, A 0.000, B 0.000, C 0.000 }
gfCNCPoint5[15561] = {X 1.6856, Y 9.3503, Z -7.1667, A 0.000, B 0.000, C 0.000 }
gfCNCPoint5[15562] = {X 2.6032, Y 9.6032, Z -7.1667, A 0.000, B 0.000, C 0.000 }
gfCNCPoint5[15563] = {X 3.5209, Y 9.1926, Z -7.1667, A 0.000, B 0.000, C 0.000 }
gfCNCPoint5[15564] = {X 5.5908, Y 8.4128, Z -7.1667, A 0.000, B 0.000, C 0.000 }
gfCNCPoint5[15565] = {X 7.7244, Y 7.8291, Z -7.1667, A 0.000, B 0.000, C 0.000 }
gfCNCPoint5[15566] = {X 9.9031, Y 7.4467, Z -7.1667, A 0.000, B 0.000, C 0.000 }
gfCNCPoint5[15567] = {X 12.1079, Y 7.2688, Z -7.1667, A 0.000, B 0.000, C 0.000 }
gfCNCPoint5[15568] = {X 14.3197, Y 7.2972, Z -7.1667, A 0.000, B 0.000, C 0.000 }
gfCNCPoint5[15569] = {X 16.5192, Y 7.5314, Z -7.1667, A 0.000, B 0.000, C 0.000 }
gfCNCPoint5[15570] = {X 18.2466, Y 7.8851, Z -7.1667, A 0.000, B 0.000, C 0.000 }
gfCNCPoint5[15571] = {X 19.9292, Y 8.4122, Z -7.1667, A 0.000, B 0.000, C 0.000 }
gfCNCPoint5[15572] = {X 21.5497, Y 9.1072, Z -7.1667, A 0.000, B 0.000, C 0.000 }
gfCNCPoint5[15573] = {X 23.0914, Y 9.9629, Z -7.1667, A 0.000, B 0.000, C 0.000 }
gfCNCPoint5[15574] = {X 24.5384, Y 10.9706, Z -7.1667, A 0.000, B 0.000, C 0.000 }
gfCNCPoint5[15575] = {X 25.6171, Y 11.9138, Z -7.1667, A 0.000, B 0.000, C 0.000 }
gfCNCPoint5[15576] = {X 26.5847, Y 12.9707, Z -7.1667, A 0.000, B 0.000, C 0.000 }
gfCNCPoint5[15577] = {X 27.4294, Y 14.1281, Z -7.1667, A 0.000, B 0.000, C 0.000 }
gfCNCPoint5[15578] = {X 28.1408, Y 15.3720, Z -7.1667, A 0.000, B 0.000, C 0.000 }
gfCNCPoint5[15579] = {X 28.7101, Y 16.6870, Z -7.1667, A 0.000, B 0.000, C 0.000 }
gfCNCPoint5[15580] = {X 29.1822, Y 18.3342, Z -7.1667, A 0.000, B 0.000, C 0.000 }
gfCNCPoint5[15581] = {X 29.4623, Y 20.0247, Z -7.1667, A 0.000, B 0.000, C 0.000 }
gfCNCPoint5[15582] = {X 29.5468, Y 21.7361, Z -7.1667, A 0.000, B 0.000, C 0.000 }
gfCNCPoint5[15583] = {X 29.4345, Y 23.4459, Z -7.1667, A 0.000, B 0.000, C 0.000 }
gfCNCPoint5[15584] = {X 29.1271, Y 25.1316, Z -7.1667, A 0.000, B 0.000, C 0.000 }
gfCNCPoint5[15585] = {X 28.6977, Y 26.5415, Z -7.1667, A 0.000, B 0.000, C 0.000 }
gfCNCPoint5[15586] = {X 28.0933, Y 27.8857, Z -7.1667, A 0.000, B 0.000, C 0.000 }
gfCNCPoint5[15587] = {X 27.3235, Y 29.1425, Z -7.1667, A 0.000, B 0.000, C 0.000 }
gfCNCPoint5[15588] = {X 26.4008, Y 30.2917, Z -7.1667, A 0.000, B 0.000, C 0.000 }
gfCNCPoint5[15589] = {X 25.3399, Y 31.3148, Z -7.1667, A 0.000, B 0.000, C 0.000 }
gfCNCPoint5[15590] = {X 25.2272, Y 31.4092, Z -7.1667, A 0.000, B 0.000, C 0.000 }
gfCNCPoint5[15591] = {X 25.1134, Y 31.5021, Z -7.1667, A 0.000, B 0.000, C 0.000 }
gfCNCPoint5[15592] = {X 25.9473, Y 31.8269, Z -7.1667, A 0.000, B 0.000, C 0.000 }
gfCNCPoint5[15593] = {X 26.6945, Y 32.3194, Z -7.1667, A 0.000, B 0.000, C 0.000 }
gfCNCPoint5[15594] = {X 27.3217, Y 32.9578, Z -7.1667, A 0.000, B 0.000, C 0.000 }
gfCNCPoint5[15595] = {X 27.8009, Y 33.7136, Z -7.1667, A 0.000, B 0.000, C 0.000 }
gfCNCPoint5[15596] = {X 30.8380, Y 39.9879, Z -7.1667, A 0.000, B 0.000, C 0.000 }
gfCNCPoint5[15597] = {X 31.1526, Y 40.8802, Z -7.1667, A 0.000, B 0.000, C 0.000 }
gfCNCPoint5[15598] = {X 31.2615, Y 41.8200, Z -7.1667, A 0.000, B 0.000, C 0.000 }
gfCNCPoint5[15599] = {X 31.1593, Y 42.7606, Z -7.1667, A 0.000, B 0.000, C 0.000 }
gfCNCPoint5[15600] = {X 30.8511, Y 43.6551, Z -7.1667, A 0.000, B 0.000, C 0.000 }
gfCNCPoint5[15601] = {X 30.3522, Y 44.4590, Z -7.1667, A 0.000, B 0.000, C 0.000 }
gfCNCPoint5[15602] = {X 29.6874, Y 45.1323, Z -7.1667, A 0.000, B 0.000, C 0.000 }
gfCNCPoint5[15603] = {X 29.1514, Y 45.5656, Z -7.1667, A 0.000, B 0.000, C 0.000 }
gfCNCPoint5[15604] = {X 28.4546, Y 46.0241, Z -7.1667, A 0.000, B 0.000, C 0.000 }
gfCNCPoint5[15605] = {X 27.6816, Y 46.3376, Z -7.1667, A 0.000, B 0.000, C 0.000 }
gfCNCPoint5[15606] = {X 26.8622, Y 46.4941, Z -7.1667, A 0.000, B 0.000, C 0.000 }
gfCNCPoint5[15607] = {X 26.0281, Y 46.4876, Z -7.1667, A 0.000, B 0.000, C 0.000 }
gfCNCPoint5[15608] = {X 25.2113, Y 46.3183, Z -7.1667, A 0.000, B 0.000, C 0.000 }
gfCNCPoint5[15609] = {X 23.4064, Y 47.2731, Z -7.1667, A 0.000, B 0.000, C 0.000 }
gfCNCPoint5[15610] = {X 21.5390, Y 48.0991, Z -7.1667, A 0.000, B 0.000, C 0.000 }
gfCNCPoint5[15611] = {X 19.6184, Y 48.7923, Z -7.1667, A 0.000, B 0.000, C 0.000 }
gfCNCPoint5[15612] = {X 17.6854, Y 49.3379, Z -7.1667, A 0.000, B 0.000, C 0.000 }
gfCNCPoint5[15613] = {X 15.7118, Y 49.7103, Z -7.1667, A 0.000, B 0.000, C 0.000 }
gfCNCPoint5[15614] = {X 13.7129, Y 49.9066, Z -7.1667, A 0.000, B 0.000, C 0.000 }
gfCNCPoint5[15615] = {X 11.7045, Y 49.9253, Z -7.1667, A 0.000, B 0.000, C 0.000 }
gfCNCPoint5[15616] = {X 9.7024, Y 49.7662, Z -7.1667, A 0.000, B 0.000, C 0.000 }
gfCNCPoint5[15617] = {X 7.7221, Y 49.4305, Z -7.1667, A 0.000, B 0.000, C 0.000 }
gfCNCPoint5[15618] = {X 5.8297, Y 48.9121, Z -7.1667, A 0.000, B 0.000, C 0.000 }
gfCNCPoint5[15619] = {X 4.0114, Y 48.1744, Z -7.1667, A 0.000, B 0.000, C 0.000 }
gfCNCPoint5[15620] = {X 2.2927, Y 47.2278, Z -7.1667, A 0.000, B 0.000, C 0.000 }
gfCNCPoint5[15621] = {X 0.6973, Y 46.0854, Z -7.1667, A 0.000, B 0.000, C 0.000 }
gfCNCPoint5[15622] = {X -0.4280, Y 45.0737, Z -7.1667, A 0.000, B 0.000, C 0.000 }
gfCNCPoint5[15623] = {X -1.4275, Y 43.9376, Z -7.1667, A 0.000, B 0.000, C 0.000 }
gfCNCPoint5[15624] = {X -2.2876, Y 42.6926, Z -7.1667, A 0.000, B 0.000, C 0.000 }
gfCNCPoint5[15625] = {X -2.9965, Y 41.3557, Z -7.1667, A 0.000, B 0.000, C 0.000 }
gfCNCPoint5[15626] = {X -3.5444, Y 39.9451, Z -7.1667, A 0.000, B 0.000, C 0.000 }
gfCNCPoint5[15627] = {X -3.6231, Y 39.6922, Z -7.1667, A 0.000, B 0.000, C 0.000 }
gfCNCPoint5[15628] = {X -3.6967, Y 39.4377, Z -7.1667, A 0.000, B 0.000, C 0.000 }
gfCNCPoint5[15629] = {X -4.7677, Y 35.5838, Z -7.1667, A 0.000, B 0.000, C 0.000 }
gfCNCPoint5[15630] = {X -8.0049, Y 35.6351, Z -7.1667, A 0.000, B 0.000, C 0.000 }
gfCNCPoint5[15631] = {X -8.0049, Y 35.6351, Z -4.1667, A 0.000, B 0.000, C 0.000 }
gfCNCPoint5[15632] = {X -8.0049, Y 35.6351, Z 11.0000, A 0.000, B 0.000, C 0.000 }
gfCNCPoint5[15633] = {X -7.6967, Y 17.3022, Z 11.0000, A 0.000, B 0.000, C 0.000 }
gfCNCPoint5[15634] = {X -7.6967, Y 17.3022, Z -4.1667, A 0.000, B 0.000, C 0.000 }
gfCNCPoint5[15635] = {X -7.6967, Y 17.3022, Z -7.1667, A 0.000, B 0.000, C 0.000 }
gfCNCPoint5[15636] = {X -4.2185, Y 17.3022, Z -7.1667, A 0.000, B 0.000, C 0.000 }
gfCNCPoint5[15637] = {X -3.6967, Y 13.3364, Z -7.1667, A 0.000, B 0.000, C 0.000 }
gfCNCPoint5[15638] = {X -3.6097, Y 12.8769, Z -7.1667, A 0.000, B 0.000, C 0.000 }
gfCNCPoint5[15639] = {X -3.4717, Y 12.4301, Z -7.1667, A 0.000, B 0.000, C 0.000 }
gfCNCPoint5[15640] = {X -3.0336, Y 11.5717, Z -7.1667, A 0.000, B 0.000, C 0.000 }
gfCNCPoint5[15641] = {X -2.4098, Y 10.8371, Z -7.1667, A 0.000, B 0.000, C 0.000 }
gfCNCPoint5[15642] = {X -1.6337, Y 10.2658, Z -7.1667, A 0.000, B 0.000, C 0.000 }
